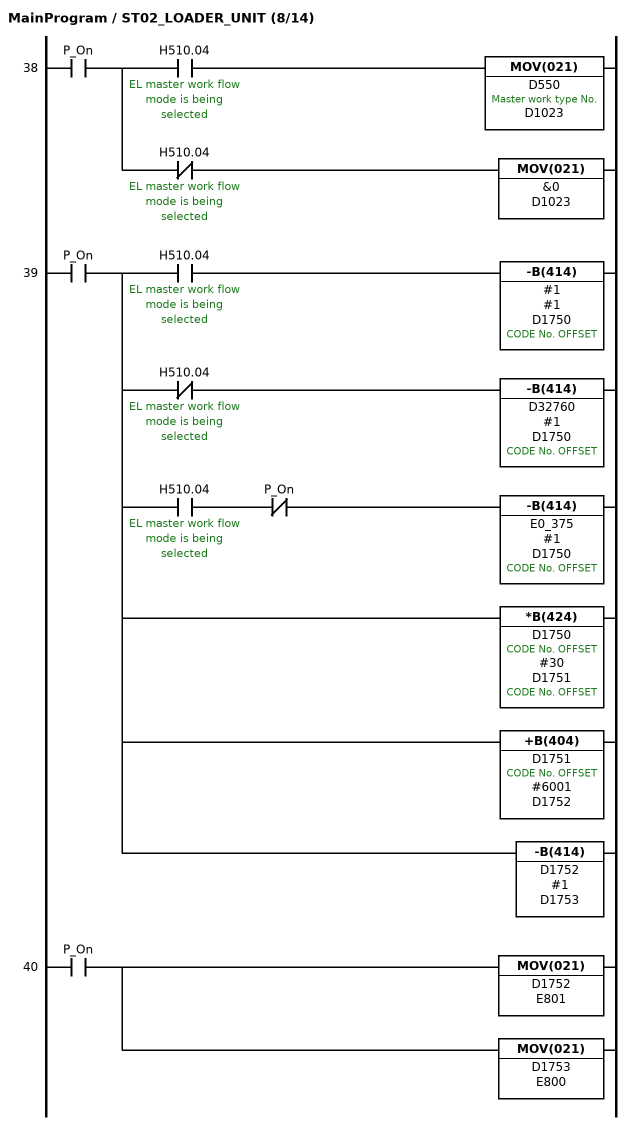
; [picture p312: MainProgram / ST02_LOADER_UNIT, rungs 38-40]
; rung 38
LD P_On
OUT TR0
AND H510.04  ; EL master work flow mode is being selected
MOV(021) D550 D1023  ; Master work type No.
LD TR0
ANDNOT H510.04  ; EL master work flow mode is being selected
MOV(021) &0 D1023
; rung 39
LD P_On
OUT TR0
AND H510.04  ; EL master work flow mode is being selected
-B(414) #1 #1 D1750  ; CODE No. OFFSET
LD TR0
ANDNOT H510.04  ; EL master work flow mode is being selected
-B(414) D32760 #1 D1750  ; CODE No. OFFSET
LD TR0
AND H510.04  ; EL master work flow mode is being selected
ANDNOT P_On
-B(414) E0_375 #1 D1750  ; CODE No. OFFSET
LD TR0
*B(424) D1750 #30 D1751  ; CODE No. OFFSET
+B(404) D1751 #6001 D1752  ; CODE No. OFFSET
-B(414) D1752 #1 D1753
; rung 40
LD P_On
MOV(021) D1752 E801
MOV(021) D1753 E800

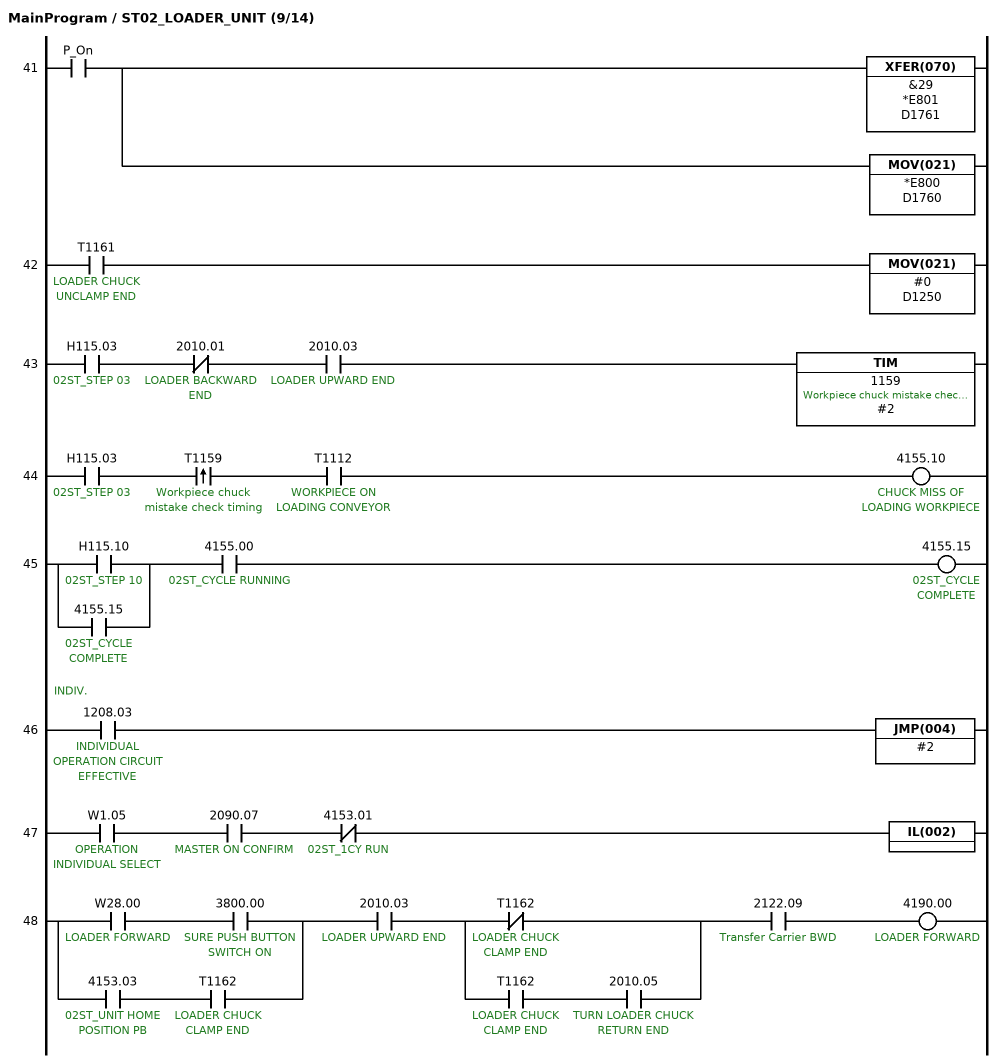
; rung 41
LD P_On
XFER(070) &29 *E801 D1761
MOV(021) *E800 D1760
; rung 42
LD T1161  ; LOADER CHUCK UNCLAMP END
MOV(021) #0 D1250
; rung 43
LD H115.03  ; 02ST_STEP 03
ANDNOT 2010.01  ; LOADER BACKWARD END
AND 2010.03  ; LOADER UPWARD END
TIM 1159 #2  ; Workpiece chuck mistake check timing
; rung 44
LD H115.03  ; 02ST_STEP 03
@AND T1159  ; Workpiece chuck mistake check timing
AND T1112  ; WORKPIECE ON LOADING CONVEYOR
OUT 4155.10  ; CHUCK MISS OF LOADING WORKPIECE
; rung 45
LD H115.10  ; 02ST_STEP 10
OR 4155.15  ; 02ST_CYCLE COMPLETE
AND 4155.00  ; 02ST_CYCLE RUNNING
OUT 4155.15  ; 02ST_CYCLE COMPLETE
; rung 46: INDIV.
LD 1208.03  ; INDIVIDUAL OPERATION CIRCUIT EFFECTIVE
JMP(004) #2
; rung 47
LD W1.05  ; OPERATION INDIVIDUAL SELECT
AND 2090.07  ; MASTER ON CONFIRM
ANDNOT 4153.01  ; 02ST_1CY RUN
IL(002)
; rung 48
LD W28.00  ; LOADER FORWARD
AND 3800.00  ; SURE PUSH BUTTON SWITCH ON
LD 4153.03  ; 02ST_UNIT HOME POSITION PB
AND T1162  ; LOADER CHUCK CLAMP END
ORLD
AND 2010.03  ; LOADER UPWARD END
LDNOT T1162  ; LOADER CHUCK CLAMP END
LD T1162  ; LOADER CHUCK CLAMP END
AND 2010.05  ; TURN LOADER CHUCK RETURN END
ORLD
ANDLD
AND 2122.09  ; Transfer Carrier BWD
OUT 4190.00  ; LOADER FORWARD

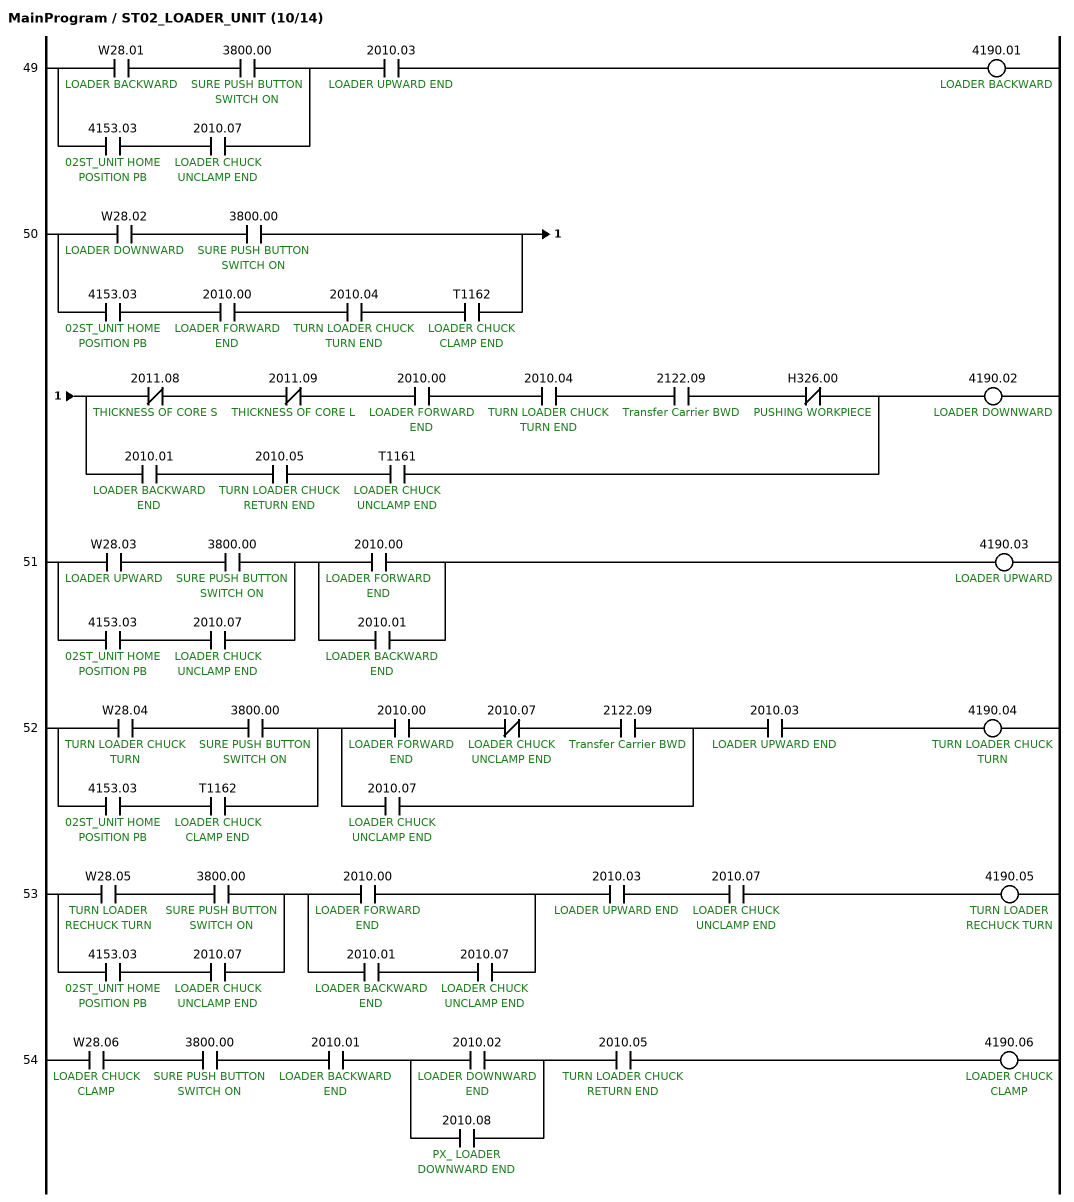
; rung 49
LD W28.01  ; LOADER BACKWARD
AND 3800.00  ; SURE PUSH BUTTON SWITCH ON
LD 4153.03  ; 02ST_UNIT HOME POSITION PB
AND 2010.07  ; LOADER CHUCK UNCLAMP END
ORLD
AND 2010.03  ; LOADER UPWARD END
OUT 4190.01  ; LOADER BACKWARD
; rung 50
LD W28.02  ; LOADER DOWNWARD
AND 3800.00  ; SURE PUSH BUTTON SWITCH ON
LD 4153.03  ; 02ST_UNIT HOME POSITION PB
AND 2010.00  ; LOADER FORWARD END
AND 2010.04  ; TURN LOADER CHUCK TURN END
AND T1162  ; LOADER CHUCK CLAMP END
ORLD
LDNOT 2011.08  ; THICKNESS OF CORE S
ANDNOT 2011.09  ; THICKNESS OF CORE L
AND 2010.00  ; LOADER FORWARD END
AND 2010.04  ; TURN LOADER CHUCK TURN END
AND 2122.09  ; Transfer Carrier BWD
ANDNOT H326.00  ; PUSHING WORKPIECE
LD 2010.01  ; LOADER BACKWARD END
AND 2010.05  ; TURN LOADER CHUCK RETURN END
AND T1161  ; LOADER CHUCK UNCLAMP END
ORLD
ANDLD
OUT 4190.02  ; LOADER DOWNWARD
; rung 51
LD W28.03  ; LOADER UPWARD
AND 3800.00  ; SURE PUSH BUTTON SWITCH ON
LD 4153.03  ; 02ST_UNIT HOME POSITION PB
AND 2010.07  ; LOADER CHUCK UNCLAMP END
ORLD
LD 2010.00  ; LOADER FORWARD END
OR 2010.01  ; LOADER BACKWARD END
ANDLD
OUT 4190.03  ; LOADER UPWARD
; rung 52
LD W28.04  ; TURN LOADER CHUCK TURN
AND 3800.00  ; SURE PUSH BUTTON SWITCH ON
LD 4153.03  ; 02ST_UNIT HOME POSITION PB
AND T1162  ; LOADER CHUCK CLAMP END
ORLD
LD 2010.00  ; LOADER FORWARD END
ANDNOT 2010.07  ; LOADER CHUCK UNCLAMP END
AND 2122.09  ; Transfer Carrier BWD
OR 2010.07  ; LOADER CHUCK UNCLAMP END
ANDLD
AND 2010.03  ; LOADER UPWARD END
OUT 4190.04  ; TURN LOADER CHUCK TURN
; rung 53
LD W28.05  ; TURN LOADER RECHUCK TURN
AND 3800.00  ; SURE PUSH BUTTON SWITCH ON
LD 4153.03  ; 02ST_UNIT HOME POSITION PB
AND 2010.07  ; LOADER CHUCK UNCLAMP END
ORLD
LD 2010.00  ; LOADER FORWARD END
LD 2010.01  ; LOADER BACKWARD END
AND 2010.07  ; LOADER CHUCK UNCLAMP END
ORLD
ANDLD
AND 2010.03  ; LOADER UPWARD END
AND 2010.07  ; LOADER CHUCK UNCLAMP END
OUT 4190.05  ; TURN LOADER RECHUCK TURN
; rung 54
LD W28.06  ; LOADER CHUCK CLAMP
AND 3800.00  ; SURE PUSH BUTTON SWITCH ON
AND 2010.01  ; LOADER BACKWARD END
LD 2010.02  ; LOADER DOWNWARD END
OR 2010.08  ; PX_ LOADER DOWNWARD END
ANDLD
AND 2010.05  ; TURN LOADER CHUCK RETURN END
OUT 4190.06  ; LOADER CHUCK CLAMP

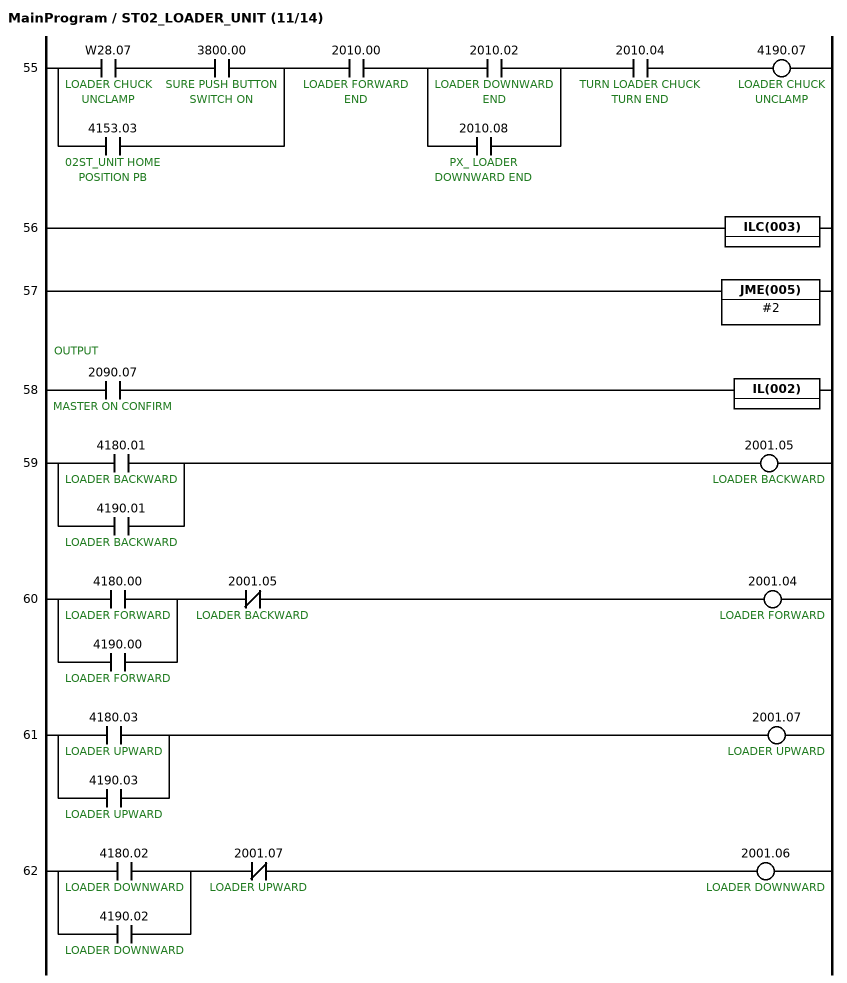
; rung 55
LD W28.07  ; LOADER CHUCK UNCLAMP
AND 3800.00  ; SURE PUSH BUTTON SWITCH ON
OR 4153.03  ; 02ST_UNIT HOME POSITION PB
AND 2010.00  ; LOADER FORWARD END
LD 2010.02  ; LOADER DOWNWARD END
OR 2010.08  ; PX_ LOADER DOWNWARD END
ANDLD
AND 2010.04  ; TURN LOADER CHUCK TURN END
OUT 4190.07  ; LOADER CHUCK UNCLAMP
; rung 56
ILC(003)
; rung 57
JME(005) #2
; rung 58: OUTPUT
LD 2090.07  ; MASTER ON CONFIRM
IL(002)
; rung 59
LD 4180.01  ; LOADER BACKWARD
OR 4190.01  ; LOADER BACKWARD
OUT 2001.05  ; LOADER BACKWARD
; rung 60
LD 4180.00  ; LOADER FORWARD
OR 4190.00  ; LOADER FORWARD
ANDNOT 2001.05  ; LOADER BACKWARD
OUT 2001.04  ; LOADER FORWARD
; rung 61
LD 4180.03  ; LOADER UPWARD
OR 4190.03  ; LOADER UPWARD
OUT 2001.07  ; LOADER UPWARD
; rung 62
LD 4180.02  ; LOADER DOWNWARD
OR 4190.02  ; LOADER DOWNWARD
ANDNOT 2001.07  ; LOADER UPWARD
OUT 2001.06  ; LOADER DOWNWARD

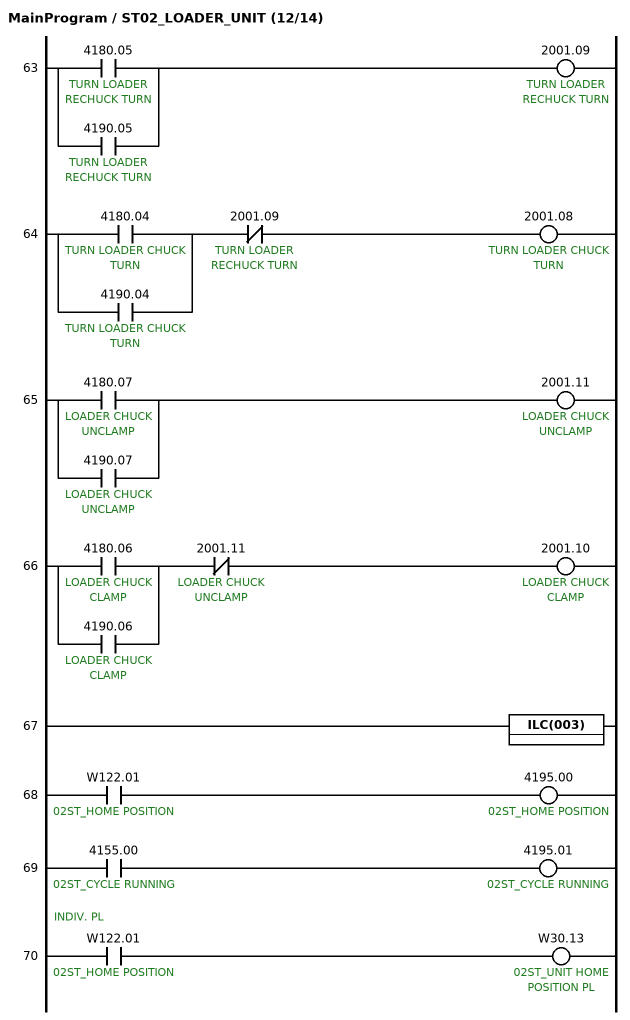
; rung 63
LD 4180.05  ; TURN LOADER RECHUCK TURN
OR 4190.05  ; TURN LOADER RECHUCK TURN
OUT 2001.09  ; TURN LOADER RECHUCK TURN
; rung 64
LD 4180.04  ; TURN LOADER CHUCK TURN
OR 4190.04  ; TURN LOADER CHUCK TURN
ANDNOT 2001.09  ; TURN LOADER RECHUCK TURN
OUT 2001.08  ; TURN LOADER CHUCK TURN
; rung 65
LD 4180.07  ; LOADER CHUCK UNCLAMP
OR 4190.07  ; LOADER CHUCK UNCLAMP
OUT 2001.11  ; LOADER CHUCK UNCLAMP
; rung 66
LD 4180.06  ; LOADER CHUCK CLAMP
OR 4190.06  ; LOADER CHUCK CLAMP
ANDNOT 2001.11  ; LOADER CHUCK UNCLAMP
OUT 2001.10  ; LOADER CHUCK CLAMP
; rung 67
ILC(003)
; rung 68
LD W122.01  ; 02ST_HOME POSITION
OUT 4195.00  ; 02ST_HOME POSITION
; rung 69
LD 4155.00  ; 02ST_CYCLE RUNNING
OUT 4195.01  ; 02ST_CYCLE RUNNING
; rung 70: INDIV. PL
LD W122.01  ; 02ST_HOME POSITION
OUT W30.13  ; 02ST_UNIT HOME POSITION PL

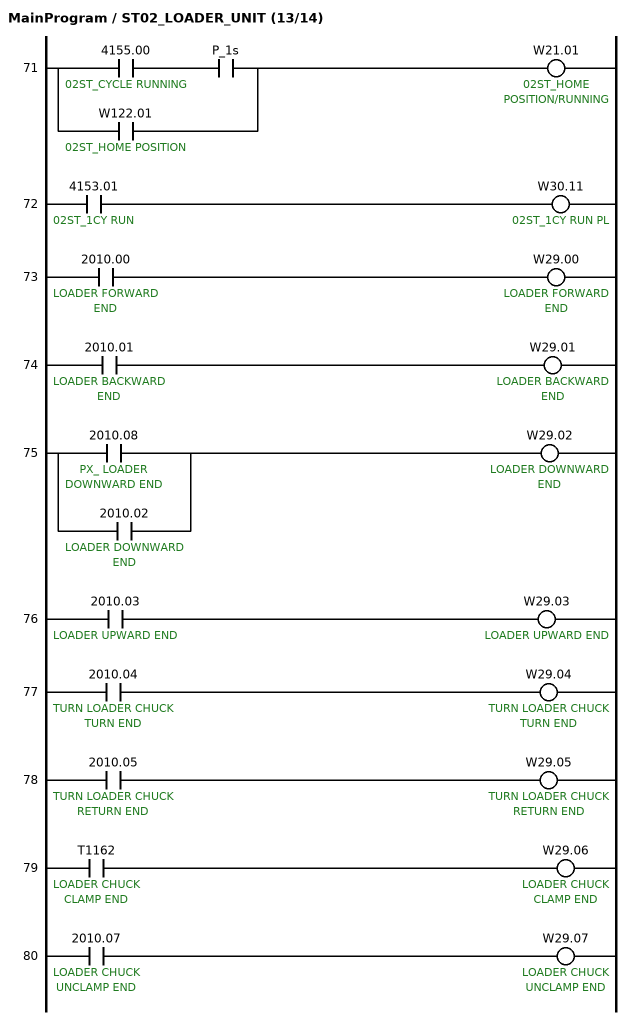
; rung 71
LD 4155.00  ; 02ST_CYCLE RUNNING
AND P_1s
OR W122.01  ; 02ST_HOME POSITION
OUT W21.01  ; 02ST_HOME POSITION/RUNNING
; rung 72
LD 4153.01  ; 02ST_1CY RUN
OUT W30.11  ; 02ST_1CY RUN PL
; rung 73
LD 2010.00  ; LOADER FORWARD END
OUT W29.00  ; LOADER FORWARD END
; rung 74
LD 2010.01  ; LOADER BACKWARD END
OUT W29.01  ; LOADER BACKWARD END
; rung 75
LD 2010.08  ; PX_ LOADER DOWNWARD END
OR 2010.02  ; LOADER DOWNWARD END
OUT W29.02  ; LOADER DOWNWARD END
; rung 76
LD 2010.03  ; LOADER UPWARD END
OUT W29.03  ; LOADER UPWARD END
; rung 77
LD 2010.04  ; TURN LOADER CHUCK TURN END
OUT W29.04  ; TURN LOADER CHUCK TURN END
; rung 78
LD 2010.05  ; TURN LOADER CHUCK RETURN END
OUT W29.05  ; TURN LOADER CHUCK RETURN END
; rung 79
LD T1162  ; LOADER CHUCK CLAMP END
OUT W29.06  ; LOADER CHUCK CLAMP END
; rung 80
LD 2010.07  ; LOADER CHUCK UNCLAMP END
OUT W29.07  ; LOADER CHUCK UNCLAMP END

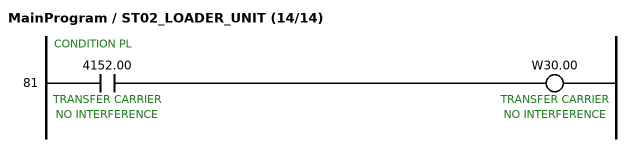
; rung 81: CONDITION PL
LD 4152.00  ; TRANSFER CARRIER NO INTERFERENCE
OUT W30.00  ; TRANSFER CARRIER NO INTERFERENCE

### Section ST03_TRANSFER_CARRIER_UNIT
; rung 0: 03ST_TRANSFER CARRIER UNIT

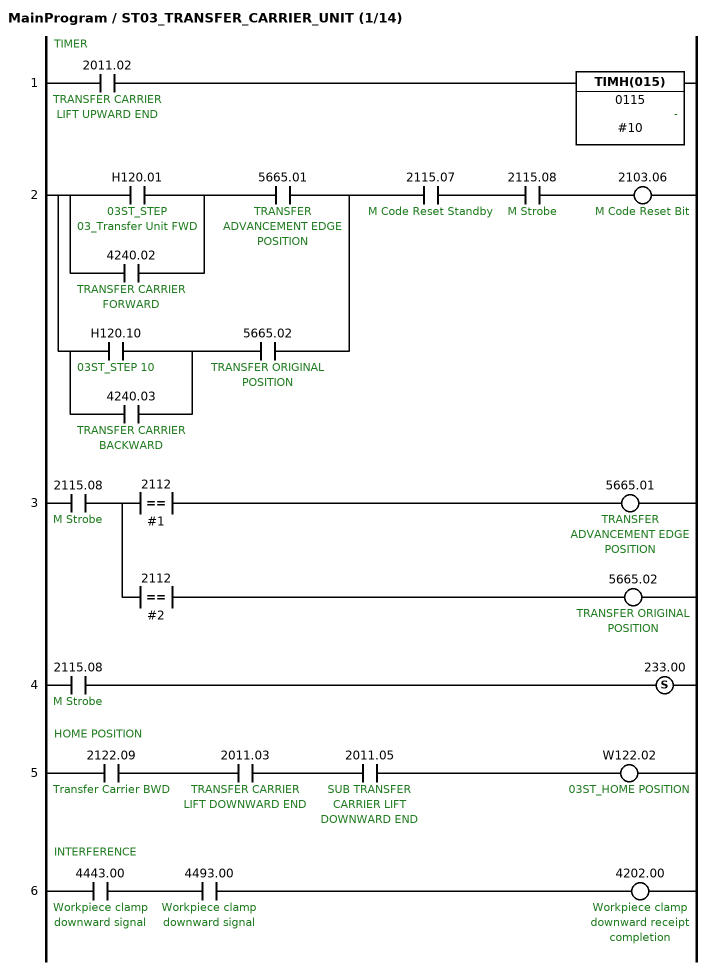
; rung 1: TIMER
LD 2011.02  ; TRANSFER CARRIER LIFT UPWARD END
TIMH(015) 0115 #10  ; -
; rung 2
LD H120.01  ; 03ST_STEP 03_Transfer Unit FWD
OR 4240.02  ; TRANSFER CARRIER FORWARD
AND 5665.01  ; TRANSFER ADVANCEMENT EDGE POSITION
LD H120.10  ; 03ST_STEP 10
OR 4240.03  ; TRANSFER CARRIER BACKWARD
AND 5665.02  ; TRANSFER ORIGINAL POSITION
ORLD
AND 2115.07  ; M Code Reset Standby
AND 2115.08  ; M Strobe
OUT 2103.06  ; M Code Reset Bit
; rung 3
LD 2115.08  ; M Strobe
OUT TR0
AND=(300) 2112 #1
OUT 5665.01  ; TRANSFER ADVANCEMENT EDGE POSITION
LD TR0
AND=(300) 2112 #2
OUT 5665.02  ; TRANSFER ORIGINAL POSITION
; rung 4
LD 2115.08  ; M Strobe
SET 233.00
; rung 5: HOME POSITION
LD 2122.09  ; Transfer Carrier BWD
AND 2011.03  ; TRANSFER CARRIER LIFT DOWNWARD END
AND 2011.05  ; SUB TRANSFER CARRIER LIFT DOWNWARD END
OUT W122.02  ; 03ST_HOME POSITION
; rung 6: INTERFERENCE
LD 4443.00  ; Workpiece clamp downward signal
AND 4493.00  ; Workpiece clamp downward signal
OUT 4202.00  ; Workpiece clamp downward receipt completion

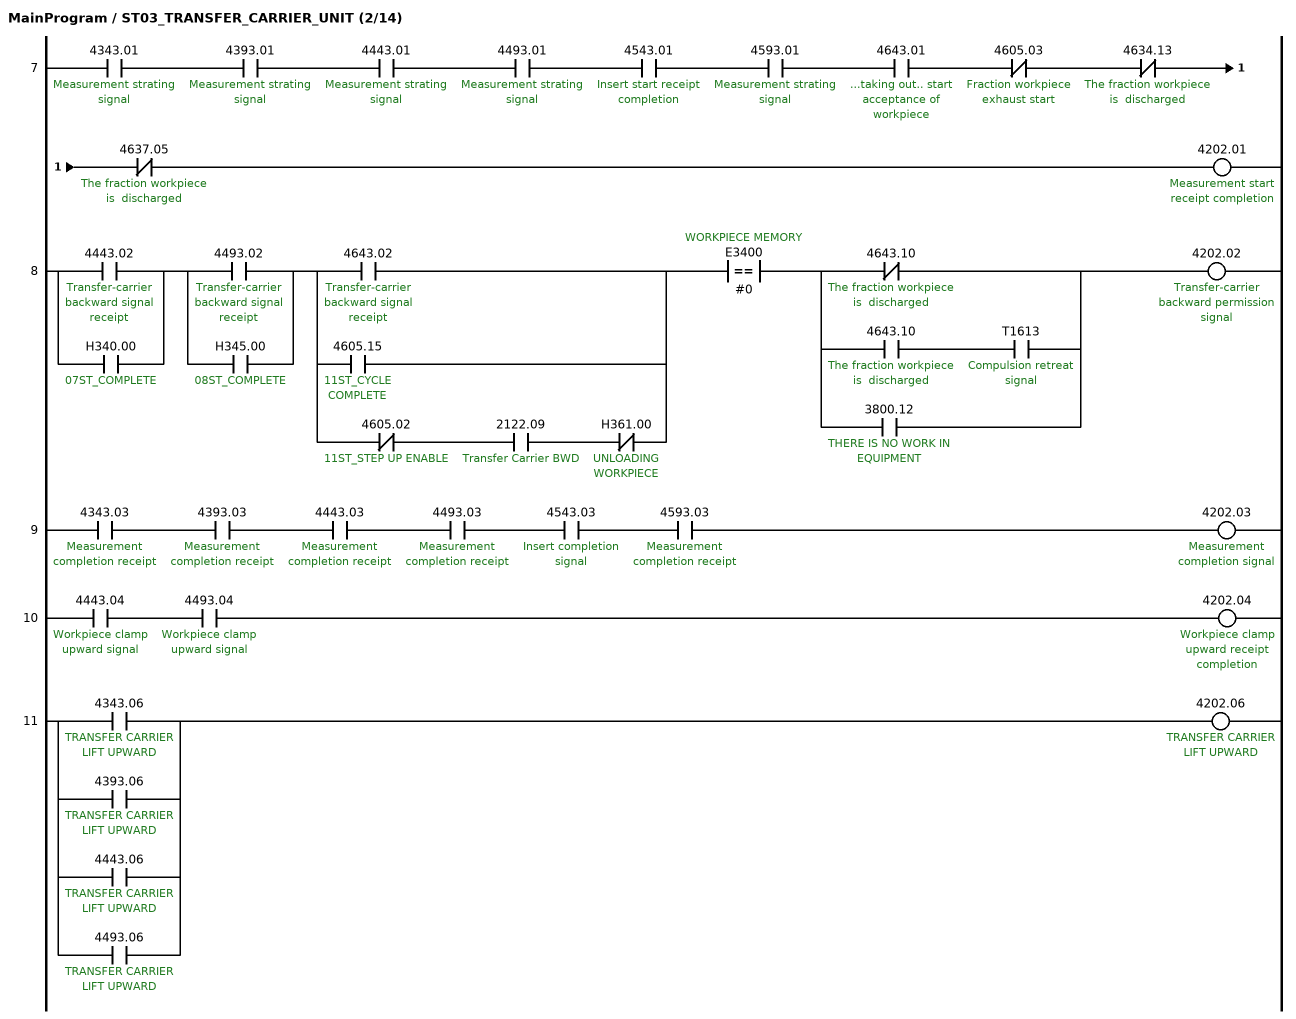
; rung 7
LD 4343.01  ; Measurement strating signal
AND 4393.01  ; Measurement strating signal
AND 4443.01  ; Measurement strating signal
AND 4493.01  ; Measurement strating signal
AND 4543.01  ; Insert start receipt completion
AND 4593.01  ; Measurement strating signal
AND 4643.01  ; ...taking out.. start acceptance of workpiece
ANDNOT 4605.03  ; Fraction workpiece exhaust start
ANDNOT 4634.13  ; The fraction workpiece is  discharged
ANDNOT 4637.05  ; The fraction workpiece is  discharged
OUT 4202.01  ; Measurement start receipt completion
; rung 8
LD 4443.02  ; Transfer-carrier backward signal receipt
OR H340.00  ; 07ST_COMPLETE
LD 4493.02  ; Transfer-carrier backward signal receipt
OR H345.00  ; 08ST_COMPLETE
ANDLD
LD 4643.02  ; Transfer-carrier backward signal receipt
OR 4605.15  ; 11ST_CYCLE COMPLETE
LDNOT 4605.02  ; 11ST_STEP UP ENABLE
AND 2122.09  ; Transfer Carrier BWD
ANDNOT H361.00  ; UNLOADING WORKPIECE
ORLD
ANDLD
AND=(300) E3400 #0  ; WORKPIECE MEMORY
LDNOT 4643.10  ; The fraction workpiece is  discharged
LD 4643.10  ; The fraction workpiece is  discharged
AND T1613  ; Compulsion retreat signal
ORLD
OR 3800.12  ; THERE IS NO WORK IN EQUIPMENT
ANDLD
OUT 4202.02  ; Transfer-carrier backward permission signal
; rung 9
LD 4343.03  ; Measurement completion receipt
AND 4393.03  ; Measurement completion receipt
AND 4443.03  ; Measurement completion receipt
AND 4493.03  ; Measurement completion receipt
AND 4543.03  ; Insert completion signal
AND 4593.03  ; Measurement completion receipt
OUT 4202.03  ; Measurement completion signal
; rung 10
LD 4443.04  ; Workpiece clamp upward signal
AND 4493.04  ; Workpiece clamp upward signal
OUT 4202.04  ; Workpiece clamp upward receipt completion
; rung 11
LD 4343.06  ; TRANSFER CARRIER LIFT UPWARD
OR 4393.06  ; TRANSFER CARRIER LIFT UPWARD
OR 4443.06  ; TRANSFER CARRIER LIFT UPWARD
OR 4493.06  ; TRANSFER CARRIER LIFT UPWARD
OUT 4202.06  ; TRANSFER CARRIER LIFT UPWARD

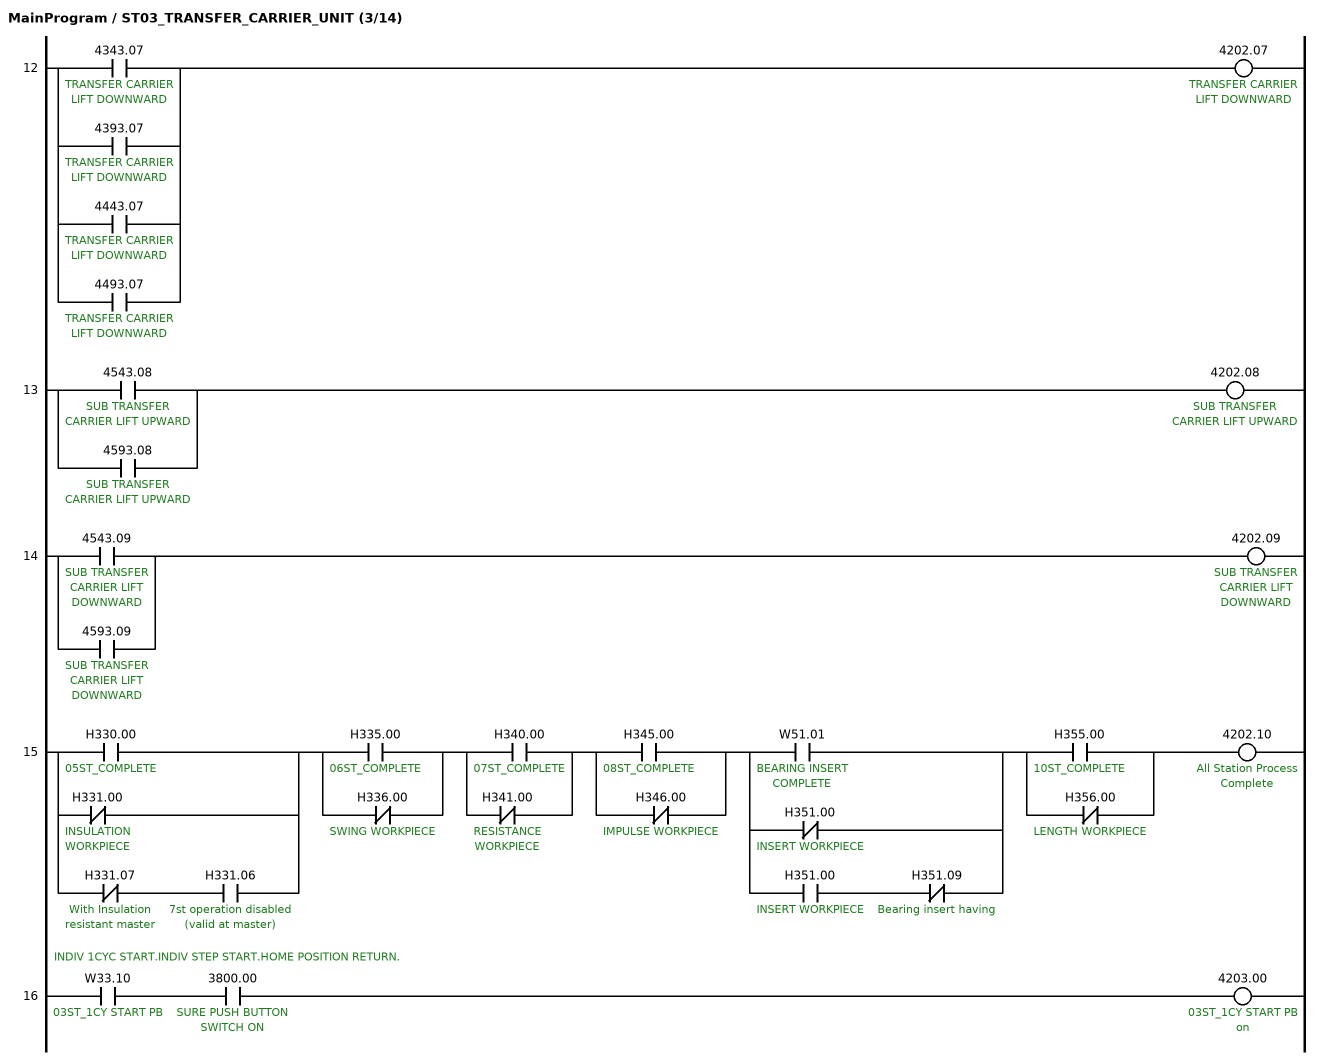
; rung 12
LD 4343.07  ; TRANSFER CARRIER LIFT DOWNWARD
OR 4393.07  ; TRANSFER CARRIER LIFT DOWNWARD
OR 4443.07  ; TRANSFER CARRIER LIFT DOWNWARD
OR 4493.07  ; TRANSFER CARRIER LIFT DOWNWARD
OUT 4202.07  ; TRANSFER CARRIER LIFT DOWNWARD
; rung 13
LD 4543.08  ; SUB TRANSFER CARRIER LIFT UPWARD
OR 4593.08  ; SUB TRANSFER CARRIER LIFT UPWARD
OUT 4202.08  ; SUB TRANSFER CARRIER LIFT UPWARD
; rung 14
LD 4543.09  ; SUB TRANSFER CARRIER LIFT DOWNWARD
OR 4593.09  ; SUB TRANSFER CARRIER LIFT DOWNWARD
OUT 4202.09  ; SUB TRANSFER CARRIER LIFT DOWNWARD
; rung 15
LD H330.00  ; 05ST_COMPLETE
ORNOT H331.00  ; INSULATION WORKPIECE
LDNOT H331.07  ; With Insulation resistant master
AND H331.06  ; 7st operation disabled (valid at master)
ORLD
LD H335.00  ; 06ST_COMPLETE
ORNOT H336.00  ; SWING WORKPIECE
ANDLD
LD H340.00  ; 07ST_COMPLETE
ORNOT H341.00  ; RESISTANCE WORKPIECE
ANDLD
LD H345.00  ; 08ST_COMPLETE
ORNOT H346.00  ; IMPULSE WORKPIECE
ANDLD
LD W51.01  ; BEARING INSERT COMPLETE
ORNOT H351.00  ; INSERT WORKPIECE
LD H351.00  ; INSERT WORKPIECE
ANDNOT H351.09  ; Bearing insert having
ORLD
ANDLD
LD H355.00  ; 10ST_COMPLETE
ORNOT H356.00  ; LENGTH WORKPIECE
ANDLD
OUT 4202.10  ; All Station Process Complete
; rung 16: INDIV 1CYC START.INDIV STEP START.HOME POSITION RETURN.
LD W33.10  ; 03ST_1CY START PB
AND 3800.00  ; SURE PUSH BUTTON SWITCH ON
OUT 4203.00  ; 03ST_1CY START PB on

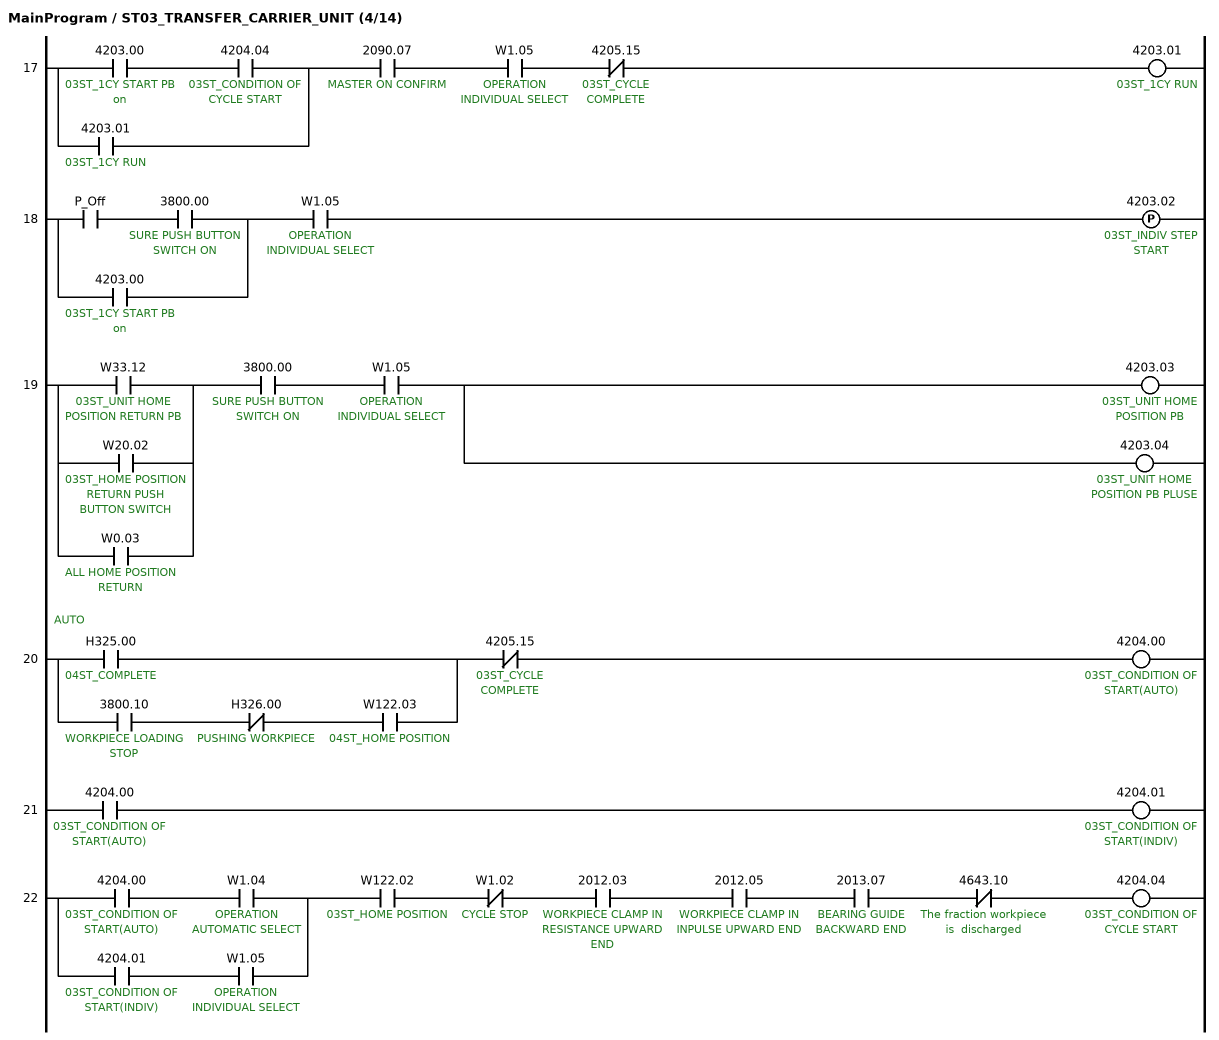
; rung 17
LD 4203.00  ; 03ST_1CY START PB on
AND 4204.04  ; 03ST_CONDITION OF CYCLE START
OR 4203.01  ; 03ST_1CY RUN
AND 2090.07  ; MASTER ON CONFIRM
AND W1.05  ; OPERATION INDIVIDUAL SELECT
ANDNOT 4205.15  ; 03ST_CYCLE COMPLETE
OUT 4203.01  ; 03ST_1CY RUN
; rung 18
LD P_Off
AND 3800.00  ; SURE PUSH BUTTON SWITCH ON
OR 4203.00  ; 03ST_1CY START PB on
AND W1.05  ; OPERATION INDIVIDUAL SELECT
DIFU(013) 4203.02  ; 03ST_INDIV STEP START
; rung 19
LD W33.12  ; 03ST_UNIT HOME POSITION RETURN PB
OR W20.02  ; 03ST_HOME POSITION RETURN PUSH BUTTON SWITCH
OR W0.03  ; ALL HOME POSITION RETURN
AND 3800.00  ; SURE PUSH BUTTON SWITCH ON
AND W1.05  ; OPERATION INDIVIDUAL SELECT
OUT 4203.03  ; 03ST_UNIT HOME POSITION PB
OUT 4203.04  ; 03ST_UNIT HOME POSITION PB PLUSE
; rung 20: AUTO
LD H325.00  ; 04ST_COMPLETE
LD 3800.10  ; WORKPIECE LOADING STOP
ANDNOT H326.00  ; PUSHING WORKPIECE
AND W122.03  ; 04ST_HOME POSITION
ORLD
ANDNOT 4205.15  ; 03ST_CYCLE COMPLETE
OUT 4204.00  ; 03ST_CONDITION OF START(AUTO)
; rung 21
LD 4204.00  ; 03ST_CONDITION OF START(AUTO)
OUT 4204.01  ; 03ST_CONDITION OF START(INDIV)
; rung 22
LD 4204.00  ; 03ST_CONDITION OF START(AUTO)
AND W1.04  ; OPERATION AUTOMATIC SELECT
LD 4204.01  ; 03ST_CONDITION OF START(INDIV)
AND W1.05  ; OPERATION INDIVIDUAL SELECT
ORLD
AND W122.02  ; 03ST_HOME POSITION
ANDNOT W1.02  ; CYCLE STOP
AND 2012.03  ; WORKPIECE CLAMP IN RESISTANCE UPWARD END
AND 2012.05  ; WORKPIECE CLAMP IN INPULSE UPWARD END
AND 2013.07  ; BEARING GUIDE BACKWARD END
ANDNOT 4643.10  ; The fraction workpiece is  discharged
OUT 4204.04  ; 03ST_CONDITION OF CYCLE START

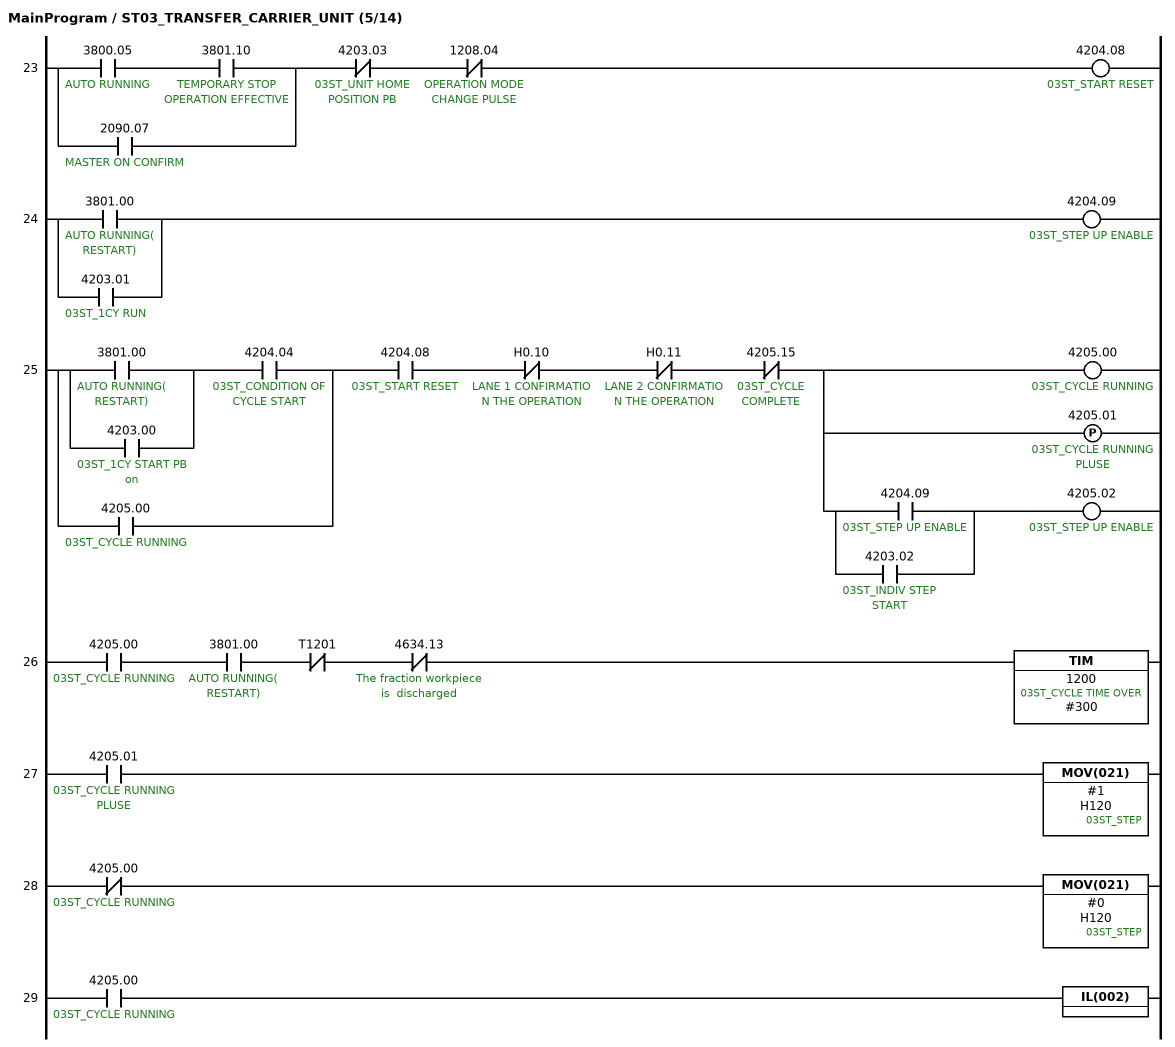
; rung 23
LD 3800.05  ; AUTO RUNNING
AND 3801.10  ; TEMPORARY STOP OPERATION EFFECTIVE
OR 2090.07  ; MASTER ON CONFIRM
ANDNOT 4203.03  ; 03ST_UNIT HOME POSITION PB
ANDNOT 1208.04  ; OPERATION MODE CHANGE PULSE
OUT 4204.08  ; 03ST_START RESET
; rung 24
LD 3801.00  ; AUTO RUNNING(RESTART)
OR 4203.01  ; 03ST_1CY RUN
OUT 4204.09  ; 03ST_STEP UP ENABLE
; rung 25
LD 3801.00  ; AUTO RUNNING(RESTART)
OR 4203.00  ; 03ST_1CY START PB on
AND 4204.04  ; 03ST_CONDITION OF CYCLE START
OR 4205.00  ; 03ST_CYCLE RUNNING
AND 4204.08  ; 03ST_START RESET
ANDNOT H0.10  ; LANE 1 CONFIRMATION THE OPERATION
ANDNOT H0.11  ; LANE 2 CONFIRMATION THE OPERATION
ANDNOT 4205.15  ; 03ST_CYCLE COMPLETE
OUT 4205.00  ; 03ST_CYCLE RUNNING
DIFU(013) 4205.01  ; 03ST_CYCLE RUNNING PLUSE
LD 4204.09  ; 03ST_STEP UP ENABLE
OR 4203.02  ; 03ST_INDIV STEP START
ANDLD
OUT 4205.02  ; 03ST_STEP UP ENABLE
; rung 26
LD 4205.00  ; 03ST_CYCLE RUNNING
AND 3801.00  ; AUTO RUNNING(RESTART)
ANDNOT T1201
ANDNOT 4634.13  ; The fraction workpiece is  discharged
TIM 1200 #300  ; 03ST_CYCLE TIME OVER
; rung 27
LD 4205.01  ; 03ST_CYCLE RUNNING PLUSE
MOV(021) #1 H120  ; 03ST_STEP
; rung 28
LDNOT 4205.00  ; 03ST_CYCLE RUNNING
MOV(021) #0 H120  ; 03ST_STEP
; rung 29
LD 4205.00  ; 03ST_CYCLE RUNNING
IL(002)

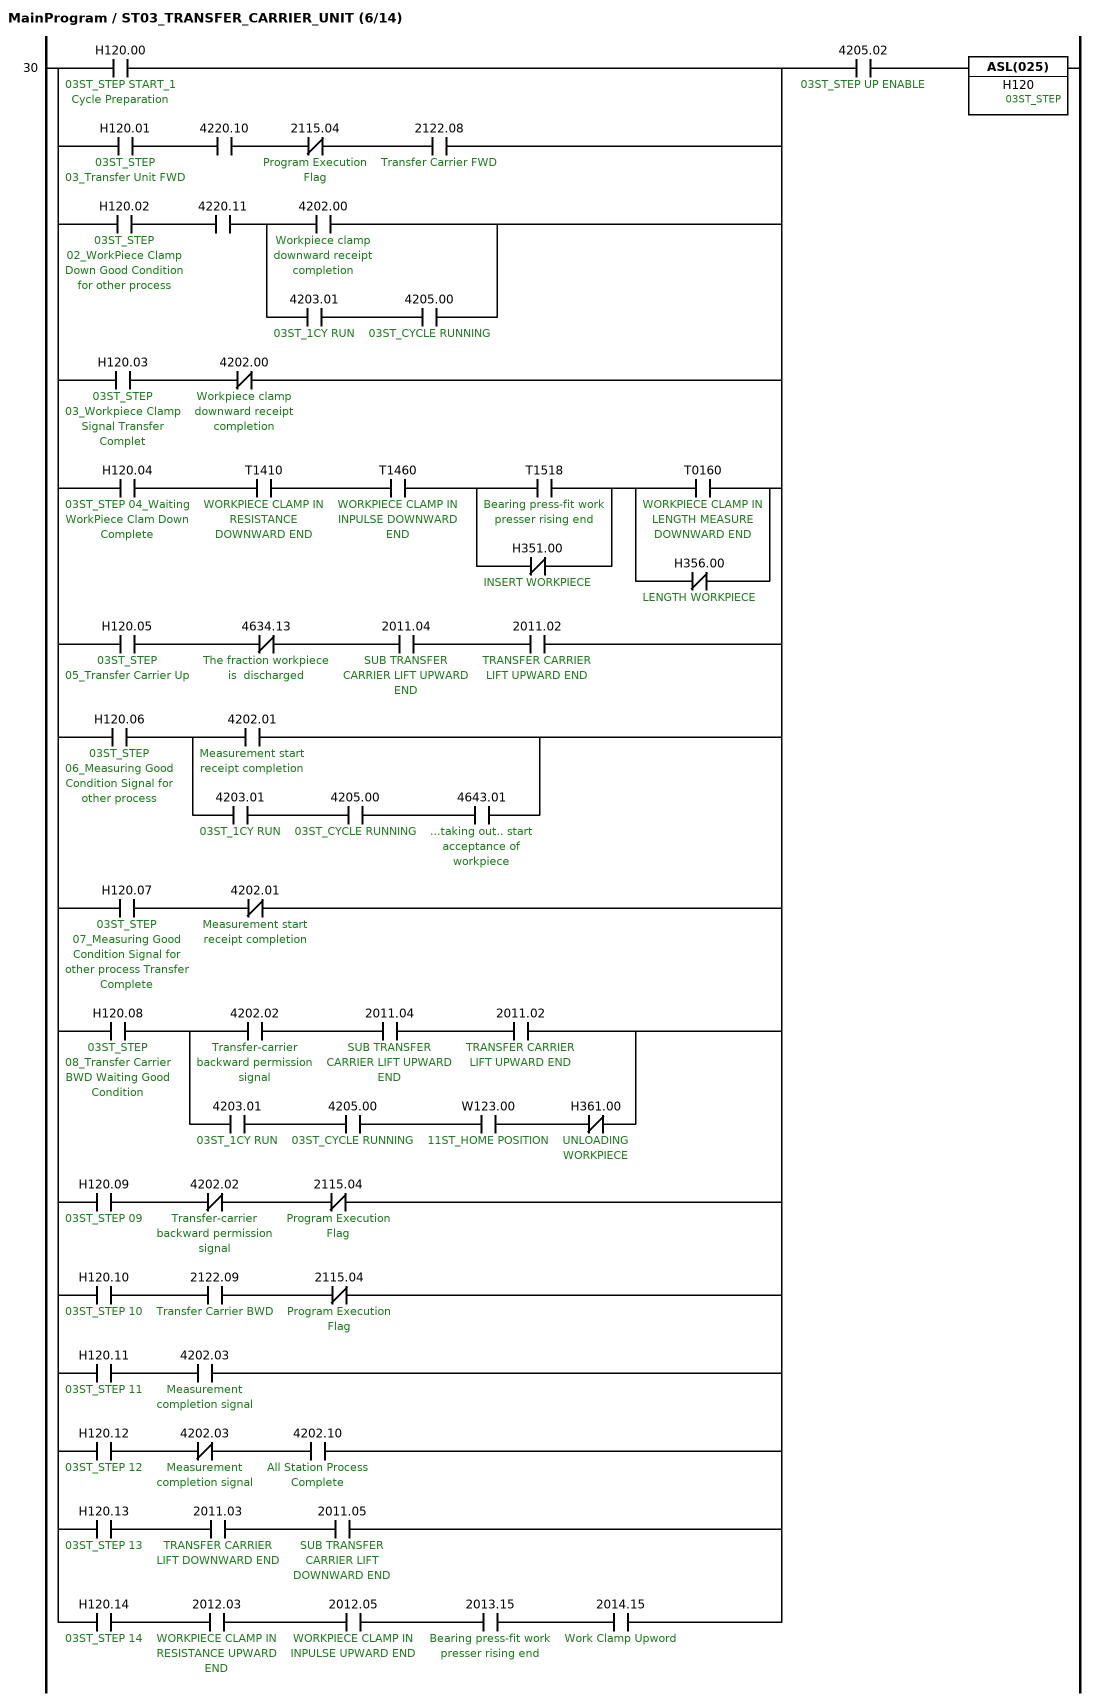
; rung 30
LD H120.00  ; 03ST_STEP START_1 Cycle Preparation
LD H120.01  ; 03ST_STEP 03_Transfer Unit FWD
AND 4220.10
ANDNOT 2115.04  ; Program Execution Flag
AND 2122.08  ; Transfer Carrier FWD
ORLD
LD H120.02  ; 03ST_STEP 02_WorkPiece Clamp Down Good Condition for other process
AND 4220.11
LD 4202.00  ; Workpiece clamp downward receipt completion
LD 4203.01  ; 03ST_1CY RUN
AND 4205.00  ; 03ST_CYCLE RUNNING
ORLD
ANDLD
ORLD
LD H120.03  ; 03ST_STEP 03_Workpiece Clamp Signal Transfer Complet
ANDNOT 4202.00  ; Workpiece clamp downward receipt completion
ORLD
LD H120.04  ; 03ST_STEP 04_Waiting WorkPiece Clam Down Complete
AND T1410  ; WORKPIECE CLAMP IN RESISTANCE DOWNWARD END
AND T1460  ; WORKPIECE CLAMP IN INPULSE DOWNWARD END
LD T1518  ; Bearing press-fit work presser rising end
ORNOT H351.00  ; INSERT WORKPIECE
ANDLD
LD T0160  ; WORKPIECE CLAMP IN LENGTH MEASURE DOWNWARD END
ORNOT H356.00  ; LENGTH WORKPIECE
ANDLD
ORLD
LD H120.05  ; 03ST_STEP 05_Transfer Carrier Up
ANDNOT 4634.13  ; The fraction workpiece is  discharged
AND 2011.04  ; SUB TRANSFER CARRIER LIFT UPWARD END
AND 2011.02  ; TRANSFER CARRIER LIFT UPWARD END
ORLD
LD H120.06  ; 03ST_STEP 06_Measuring Good Condition Signal for other process
LD 4202.01  ; Measurement start receipt completion
LD 4203.01  ; 03ST_1CY RUN
AND 4205.00  ; 03ST_CYCLE RUNNING
AND 4643.01  ; ...taking out.. start acceptance of workpiece
ORLD
ANDLD
ORLD
LD H120.07  ; 03ST_STEP 07_Measuring Good Condition Signal for other process Transfer Complete
ANDNOT 4202.01  ; Measurement start receipt completion
ORLD
LD H120.08  ; 03ST_STEP 08_Transfer Carrier BWD Waiting Good Condition
LD 4202.02  ; Transfer-carrier backward permission signal
AND 2011.04  ; SUB TRANSFER CARRIER LIFT UPWARD END
AND 2011.02  ; TRANSFER CARRIER LIFT UPWARD END
LD 4203.01  ; 03ST_1CY RUN
AND 4205.00  ; 03ST_CYCLE RUNNING
AND W123.00  ; 11ST_HOME POSITION
ANDNOT H361.00  ; UNLOADING WORKPIECE
ORLD
ANDLD
ORLD
LD H120.09  ; 03ST_STEP 09
ANDNOT 4202.02  ; Transfer-carrier backward permission signal
ANDNOT 2115.04  ; Program Execution Flag
ORLD
LD H120.10  ; 03ST_STEP 10
AND 2122.09  ; Transfer Carrier BWD
ANDNOT 2115.04  ; Program Execution Flag
ORLD
LD H120.11  ; 03ST_STEP 11
AND 4202.03  ; Measurement completion signal
ORLD
LD H120.12  ; 03ST_STEP 12
ANDNOT 4202.03  ; Measurement completion signal
AND 4202.10  ; All Station Process Complete
ORLD
LD H120.13  ; 03ST_STEP 13
AND 2011.03  ; TRANSFER CARRIER LIFT DOWNWARD END
AND 2011.05  ; SUB TRANSFER CARRIER LIFT DOWNWARD END
ORLD
LD H120.14  ; 03ST_STEP 14
AND 2012.03  ; WORKPIECE CLAMP IN RESISTANCE UPWARD END
AND 2012.05  ; WORKPIECE CLAMP IN INPULSE UPWARD END
AND 2013.15  ; Bearing press-fit work presser rising end
AND 2014.15  ; Work Clamp Upword
ORLD
AND 4205.02  ; 03ST_STEP UP ENABLE
ASL(025) H120  ; 03ST_STEP

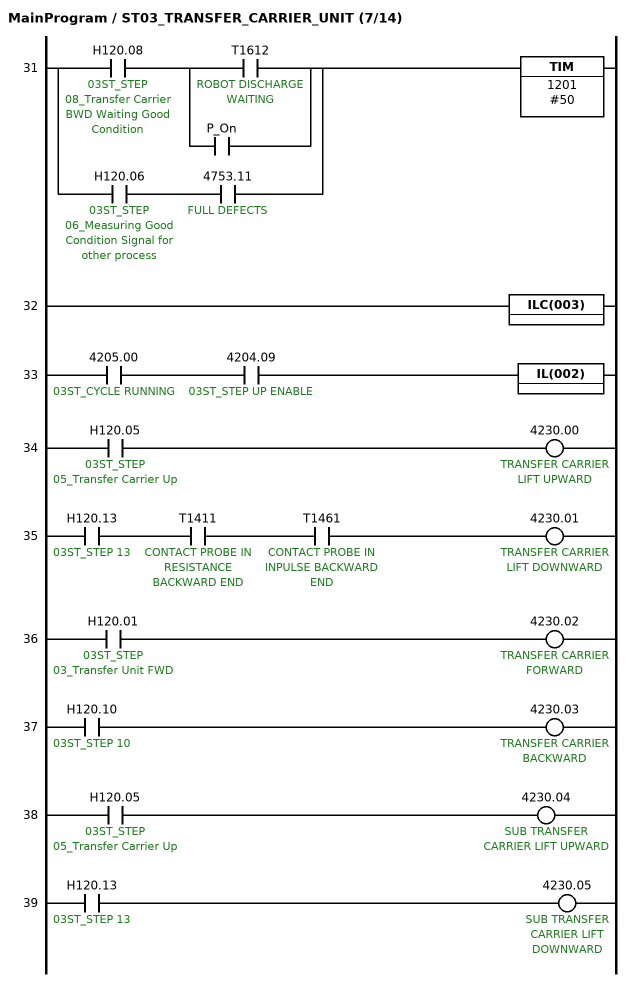
; rung 31
LD H120.08  ; 03ST_STEP 08_Transfer Carrier BWD Waiting Good Condition
LD T1612  ; ROBOT DISCHARGE WAITING
OR P_On
ANDLD
LD H120.06  ; 03ST_STEP 06_Measuring Good Condition Signal for other process
AND 4753.11  ; FULL DEFECTS
ORLD
TIM 1201 #50
; rung 32
ILC(003)
; rung 33
LD 4205.00  ; 03ST_CYCLE RUNNING
AND 4204.09  ; 03ST_STEP UP ENABLE
IL(002)
; rung 34
LD H120.05  ; 03ST_STEP 05_Transfer Carrier Up
OUT 4230.00  ; TRANSFER CARRIER LIFT UPWARD
; rung 35
LD H120.13  ; 03ST_STEP 13
AND T1411  ; CONTACT PROBE IN RESISTANCE BACKWARD END
AND T1461  ; CONTACT PROBE IN INPULSE BACKWARD END
OUT 4230.01  ; TRANSFER CARRIER LIFT DOWNWARD
; rung 36
LD H120.01  ; 03ST_STEP 03_Transfer Unit FWD
OUT 4230.02  ; TRANSFER CARRIER FORWARD
; rung 37
LD H120.10  ; 03ST_STEP 10
OUT 4230.03  ; TRANSFER CARRIER BACKWARD
; rung 38
LD H120.05  ; 03ST_STEP 05_Transfer Carrier Up
OUT 4230.04  ; SUB TRANSFER CARRIER LIFT UPWARD
; rung 39
LD H120.13  ; 03ST_STEP 13
OUT 4230.05  ; SUB TRANSFER CARRIER LIFT DOWNWARD

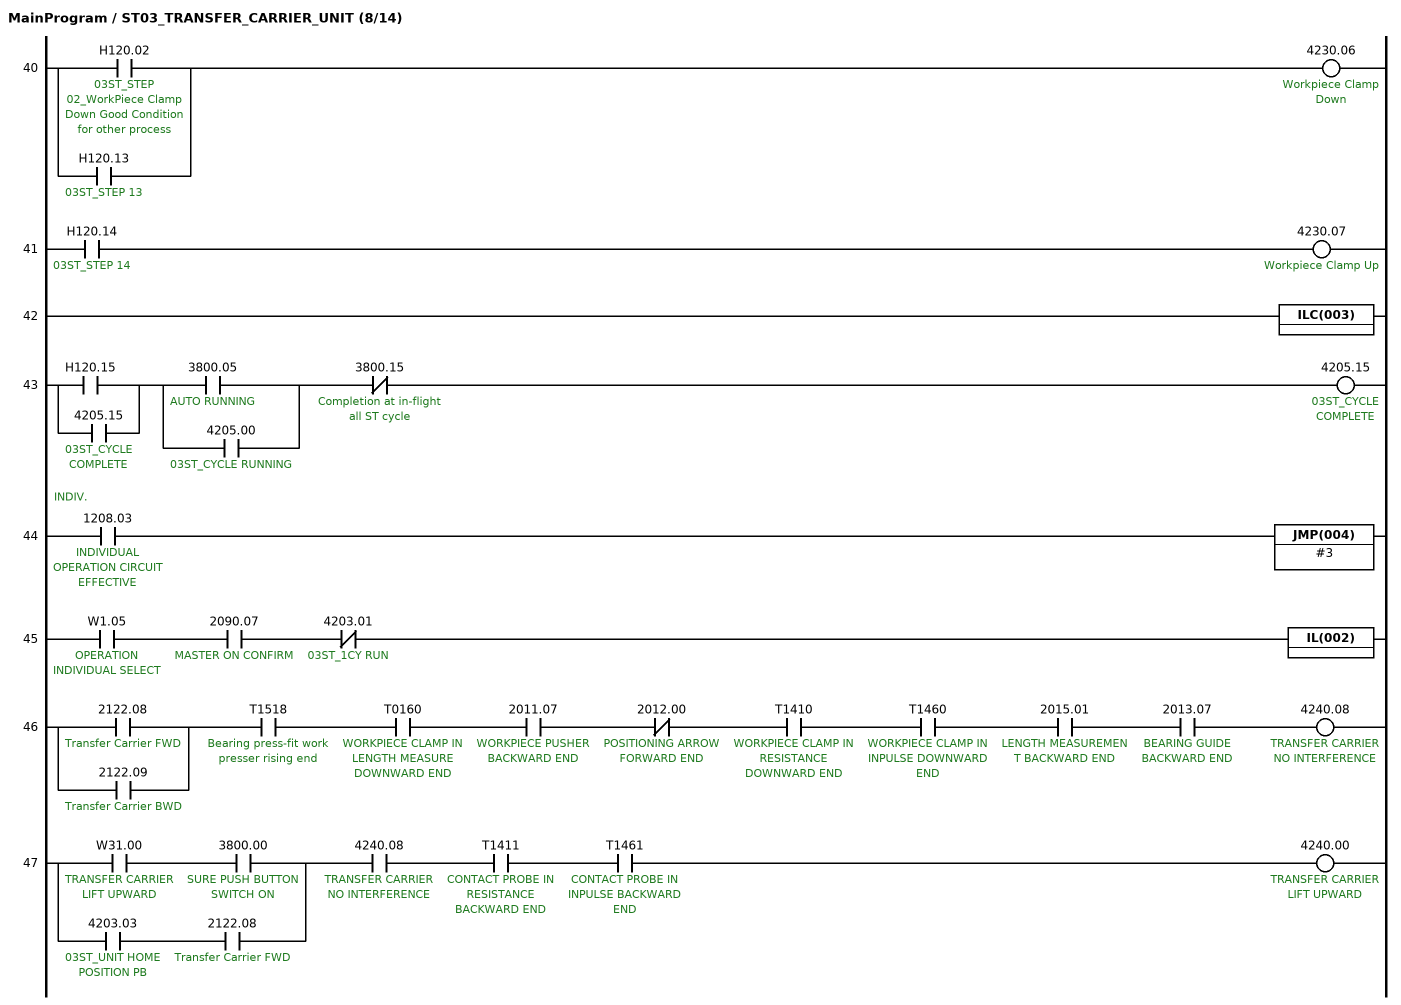
; rung 40
LD H120.02  ; 03ST_STEP 02_WorkPiece Clamp Down Good Condition for other process
OR H120.13  ; 03ST_STEP 13
OUT 4230.06  ; Workpiece Clamp Down
; rung 41
LD H120.14  ; 03ST_STEP 14
OUT 4230.07  ; Workpiece Clamp Up
; rung 42
ILC(003)
; rung 43
LD H120.15
OR 4205.15  ; 03ST_CYCLE COMPLETE
LD 3800.05  ; AUTO RUNNING
OR 4205.00  ; 03ST_CYCLE RUNNING
ANDLD
ANDNOT 3800.15  ; Completion at in-flight all ST cycle
OUT 4205.15  ; 03ST_CYCLE COMPLETE
; rung 44: INDIV.
LD 1208.03  ; INDIVIDUAL OPERATION CIRCUIT EFFECTIVE
JMP(004) #3
; rung 45
LD W1.05  ; OPERATION INDIVIDUAL SELECT
AND 2090.07  ; MASTER ON CONFIRM
ANDNOT 4203.01  ; 03ST_1CY RUN
IL(002)
; rung 46
LD 2122.08  ; Transfer Carrier FWD
OR 2122.09  ; Transfer Carrier BWD
AND T1518  ; Bearing press-fit work presser rising end
AND T0160  ; WORKPIECE CLAMP IN LENGTH MEASURE DOWNWARD END
AND 2011.07  ; WORKPIECE PUSHER BACKWARD END
ANDNOT 2012.00  ; POSITIONING ARROW FORWARD END
AND T1410  ; WORKPIECE CLAMP IN RESISTANCE DOWNWARD END
AND T1460  ; WORKPIECE CLAMP IN INPULSE DOWNWARD END
AND 2015.01  ; LENGTH MEASUREMENT BACKWARD END
AND 2013.07  ; BEARING GUIDE BACKWARD END
OUT 4240.08  ; TRANSFER CARRIER NO INTERFERENCE
; rung 47
LD W31.00  ; TRANSFER CARRIER LIFT UPWARD
AND 3800.00  ; SURE PUSH BUTTON SWITCH ON
LD 4203.03  ; 03ST_UNIT HOME POSITION PB
AND 2122.08  ; Transfer Carrier FWD
ORLD
AND 4240.08  ; TRANSFER CARRIER NO INTERFERENCE
AND T1411  ; CONTACT PROBE IN RESISTANCE BACKWARD END
AND T1461  ; CONTACT PROBE IN INPULSE BACKWARD END
OUT 4240.00  ; TRANSFER CARRIER LIFT UPWARD

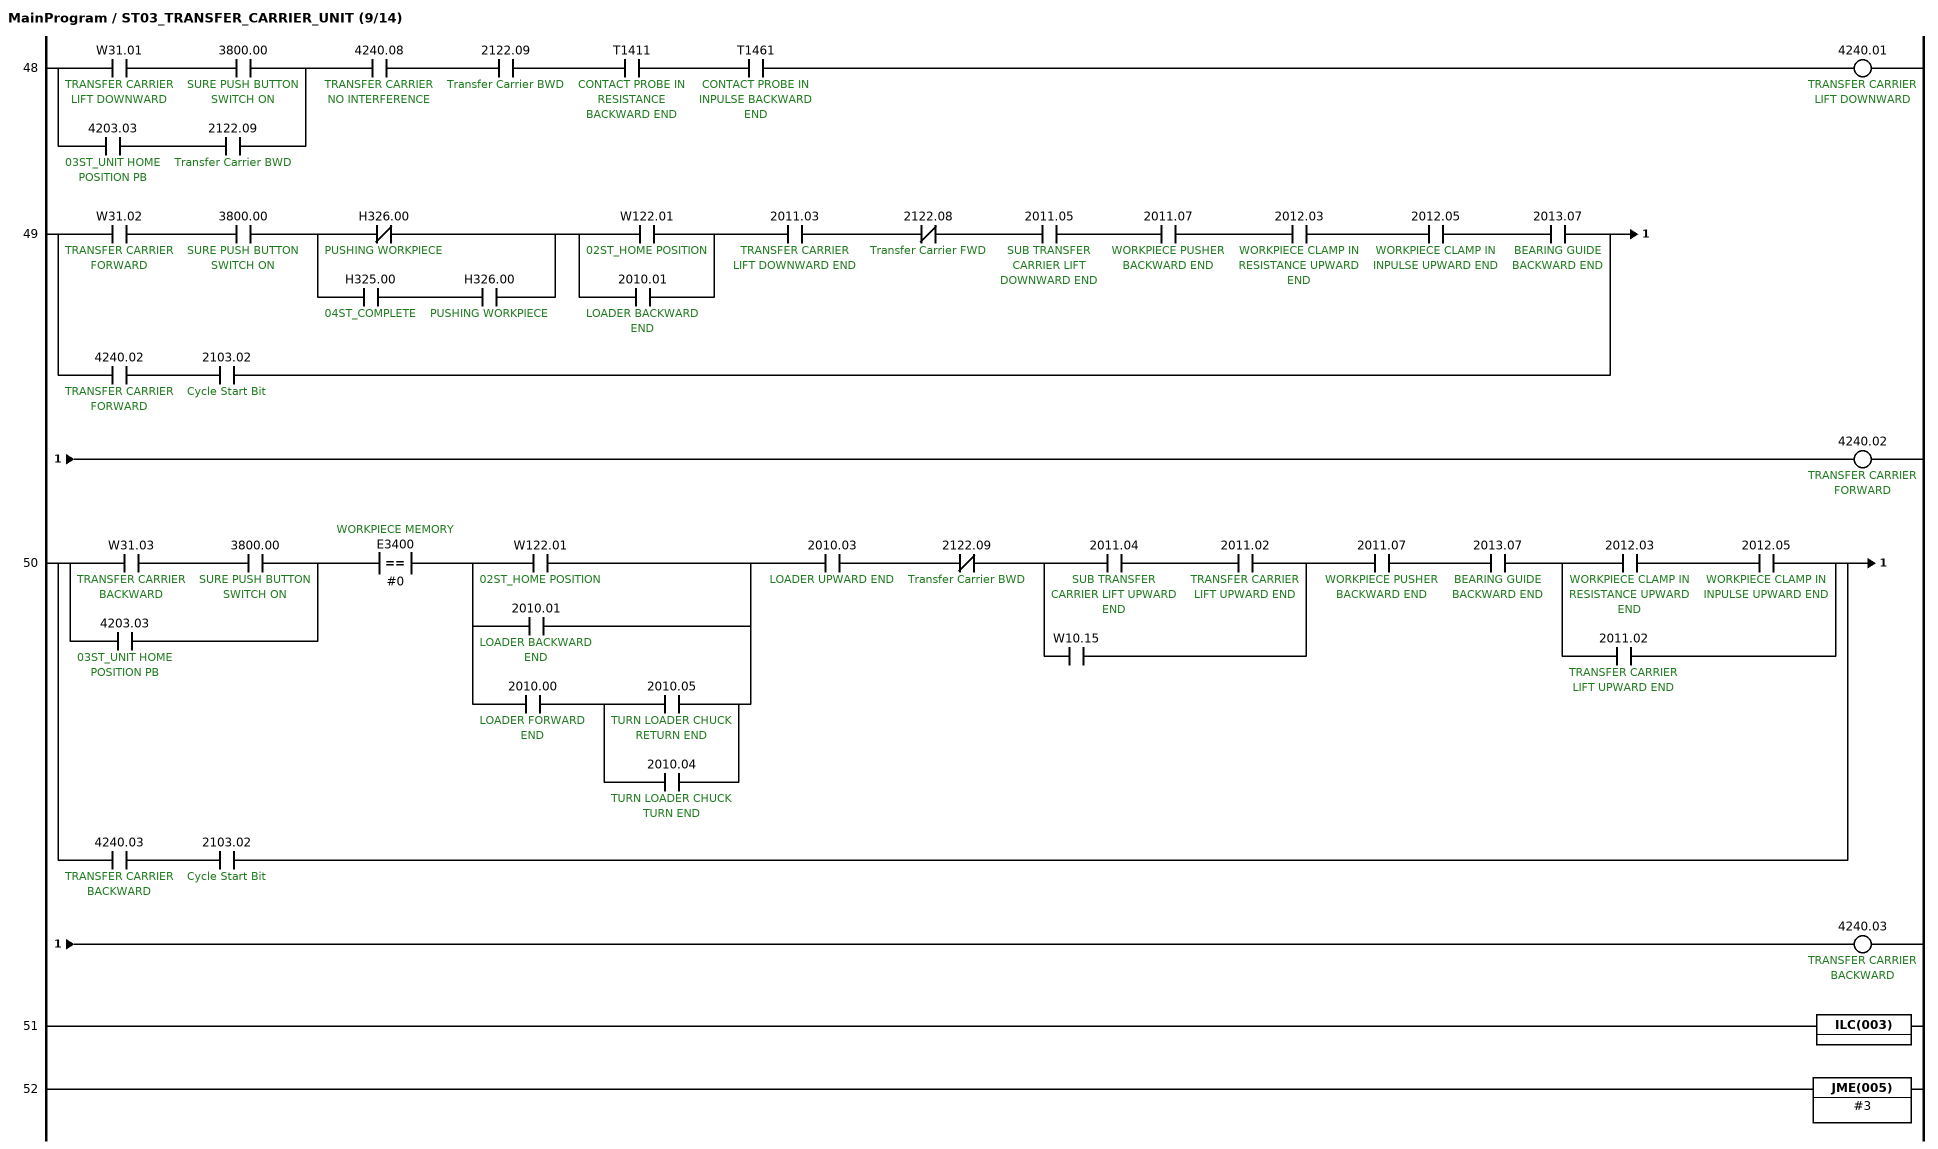
; rung 48
LD W31.01  ; TRANSFER CARRIER LIFT DOWNWARD
AND 3800.00  ; SURE PUSH BUTTON SWITCH ON
LD 4203.03  ; 03ST_UNIT HOME POSITION PB
AND 2122.09  ; Transfer Carrier BWD
ORLD
AND 4240.08  ; TRANSFER CARRIER NO INTERFERENCE
AND 2122.09  ; Transfer Carrier BWD
AND T1411  ; CONTACT PROBE IN RESISTANCE BACKWARD END
AND T1461  ; CONTACT PROBE IN INPULSE BACKWARD END
OUT 4240.01  ; TRANSFER CARRIER LIFT DOWNWARD
; rung 49
LD W31.02  ; TRANSFER CARRIER FORWARD
AND 3800.00  ; SURE PUSH BUTTON SWITCH ON
LDNOT H326.00  ; PUSHING WORKPIECE
LD H325.00  ; 04ST_COMPLETE
AND H326.00  ; PUSHING WORKPIECE
ORLD
ANDLD
LD W122.01  ; 02ST_HOME POSITION
OR 2010.01  ; LOADER BACKWARD END
ANDLD
AND 2011.03  ; TRANSFER CARRIER LIFT DOWNWARD END
ANDNOT 2122.08  ; Transfer Carrier FWD
AND 2011.05  ; SUB TRANSFER CARRIER LIFT DOWNWARD END
AND 2011.07  ; WORKPIECE PUSHER BACKWARD END
AND 2012.03  ; WORKPIECE CLAMP IN RESISTANCE UPWARD END
AND 2012.05  ; WORKPIECE CLAMP IN INPULSE UPWARD END
AND 2013.07  ; BEARING GUIDE BACKWARD END
LD 4240.02  ; TRANSFER CARRIER FORWARD
AND 2103.02  ; Cycle Start Bit
ORLD
OUT 4240.02  ; TRANSFER CARRIER FORWARD
; rung 50
LD W31.03  ; TRANSFER CARRIER BACKWARD
AND 3800.00  ; SURE PUSH BUTTON SWITCH ON
OR 4203.03  ; 03ST_UNIT HOME POSITION PB
AND=(300) E3400 #0  ; WORKPIECE MEMORY
LD W122.01  ; 02ST_HOME POSITION
OR 2010.01  ; LOADER BACKWARD END
LD 2010.00  ; LOADER FORWARD END
LD 2010.05  ; TURN LOADER CHUCK RETURN END
OR 2010.04  ; TURN LOADER CHUCK TURN END
ANDLD
ORLD
ANDLD
AND 2010.03  ; LOADER UPWARD END
ANDNOT 2122.09  ; Transfer Carrier BWD
LD 2011.04  ; SUB TRANSFER CARRIER LIFT UPWARD END
AND 2011.02  ; TRANSFER CARRIER LIFT UPWARD END
OR W10.15
ANDLD
AND 2011.07  ; WORKPIECE PUSHER BACKWARD END
AND 2013.07  ; BEARING GUIDE BACKWARD END
LD 2012.03  ; WORKPIECE CLAMP IN RESISTANCE UPWARD END
AND 2012.05  ; WORKPIECE CLAMP IN INPULSE UPWARD END
OR 2011.02  ; TRANSFER CARRIER LIFT UPWARD END
ANDLD
LD 4240.03  ; TRANSFER CARRIER BACKWARD
AND 2103.02  ; Cycle Start Bit
ORLD
OUT 4240.03  ; TRANSFER CARRIER BACKWARD
; rung 51
ILC(003)
; rung 52
JME(005) #3

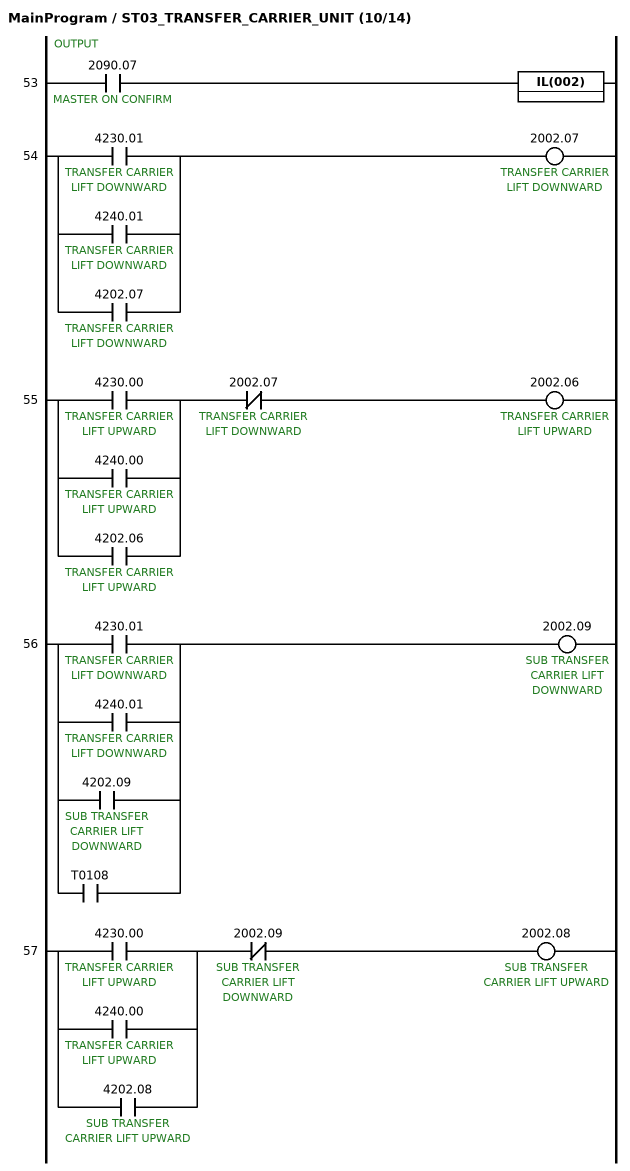
; rung 53: OUTPUT
LD 2090.07  ; MASTER ON CONFIRM
IL(002)
; rung 54
LD 4230.01  ; TRANSFER CARRIER LIFT DOWNWARD
OR 4240.01  ; TRANSFER CARRIER LIFT DOWNWARD
OR 4202.07  ; TRANSFER CARRIER LIFT DOWNWARD
OUT 2002.07  ; TRANSFER CARRIER LIFT DOWNWARD
; rung 55
LD 4230.00  ; TRANSFER CARRIER LIFT UPWARD
OR 4240.00  ; TRANSFER CARRIER LIFT UPWARD
OR 4202.06  ; TRANSFER CARRIER LIFT UPWARD
ANDNOT 2002.07  ; TRANSFER CARRIER LIFT DOWNWARD
OUT 2002.06  ; TRANSFER CARRIER LIFT UPWARD
; rung 56
LD 4230.01  ; TRANSFER CARRIER LIFT DOWNWARD
OR 4240.01  ; TRANSFER CARRIER LIFT DOWNWARD
OR 4202.09  ; SUB TRANSFER CARRIER LIFT DOWNWARD
OR T0108
OUT 2002.09  ; SUB TRANSFER CARRIER LIFT DOWNWARD
; rung 57
LD 4230.00  ; TRANSFER CARRIER LIFT UPWARD
OR 4240.00  ; TRANSFER CARRIER LIFT UPWARD
OR 4202.08  ; SUB TRANSFER CARRIER LIFT UPWARD
ANDNOT 2002.09  ; SUB TRANSFER CARRIER LIFT DOWNWARD
OUT 2002.08  ; SUB TRANSFER CARRIER LIFT UPWARD

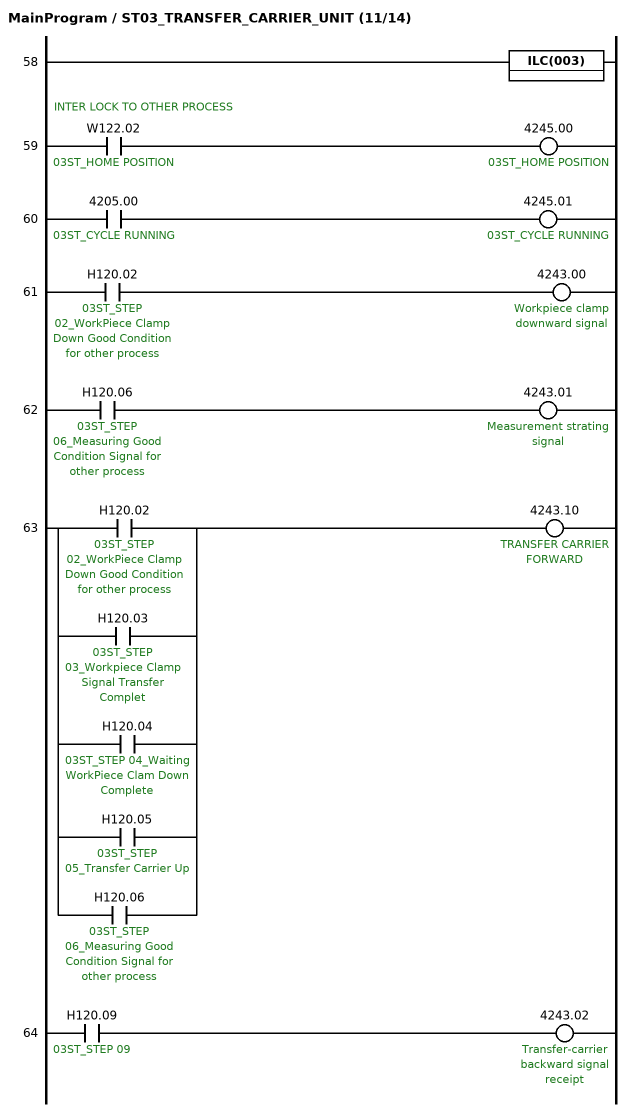
; rung 58
ILC(003)
; rung 59: INTER LOCK TO OTHER PROCESS
LD W122.02  ; 03ST_HOME POSITION
OUT 4245.00  ; 03ST_HOME POSITION
; rung 60
LD 4205.00  ; 03ST_CYCLE RUNNING
OUT 4245.01  ; 03ST_CYCLE RUNNING
; rung 61
LD H120.02  ; 03ST_STEP 02_WorkPiece Clamp Down Good Condition for other process
OUT 4243.00  ; Workpiece clamp downward signal
; rung 62
LD H120.06  ; 03ST_STEP 06_Measuring Good Condition Signal for other process
OUT 4243.01  ; Measurement strating signal
; rung 63
LD H120.02  ; 03ST_STEP 02_WorkPiece Clamp Down Good Condition for other process
OR H120.03  ; 03ST_STEP 03_Workpiece Clamp Signal Transfer Complet
OR H120.04  ; 03ST_STEP 04_Waiting WorkPiece Clam Down Complete
OR H120.05  ; 03ST_STEP 05_Transfer Carrier Up
OR H120.06  ; 03ST_STEP 06_Measuring Good Condition Signal for other process
OUT 4243.10  ; TRANSFER CARRIER FORWARD
; rung 64
LD H120.09  ; 03ST_STEP 09
OUT 4243.02  ; Transfer-carrier backward signal receipt

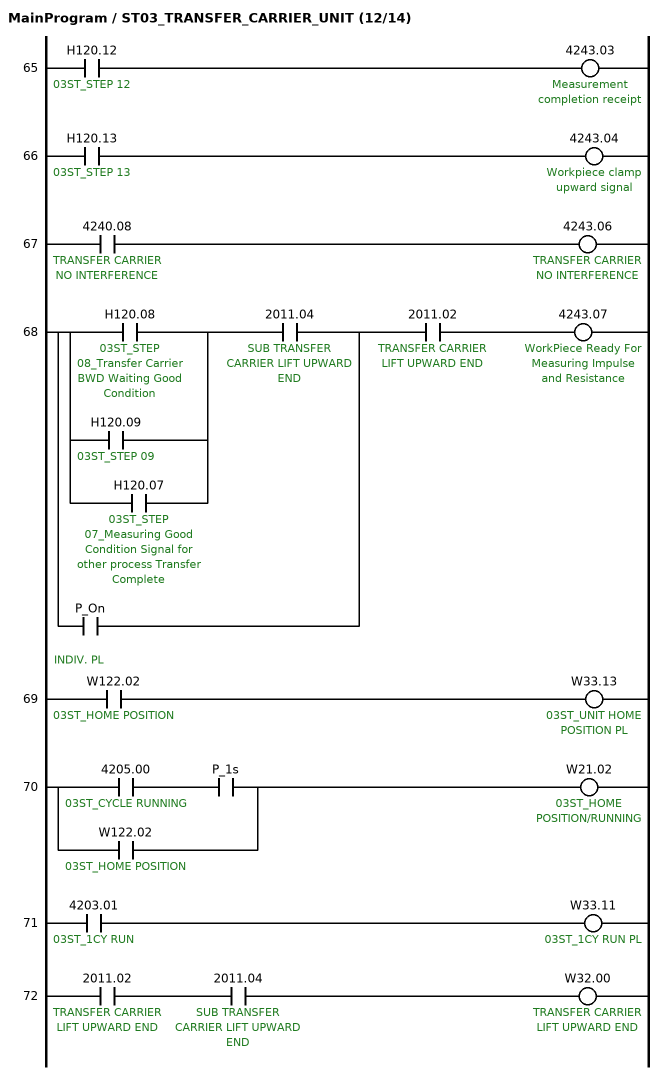
; rung 65
LD H120.12  ; 03ST_STEP 12
OUT 4243.03  ; Measurement completion receipt
; rung 66
LD H120.13  ; 03ST_STEP 13
OUT 4243.04  ; Workpiece clamp upward signal
; rung 67
LD 4240.08  ; TRANSFER CARRIER NO INTERFERENCE
OUT 4243.06  ; TRANSFER CARRIER NO INTERFERENCE
; rung 68
LD H120.08  ; 03ST_STEP 08_Transfer Carrier BWD Waiting Good Condition
OR H120.09  ; 03ST_STEP 09
OR H120.07  ; 03ST_STEP 07_Measuring Good Condition Signal for other process Transfer Complete
AND 2011.04  ; SUB TRANSFER CARRIER LIFT UPWARD END
OR P_On
AND 2011.02  ; TRANSFER CARRIER LIFT UPWARD END
OUT 4243.07  ; WorkPiece Ready For Measuring Impulse and Resistance
; rung 69: INDIV. PL
LD W122.02  ; 03ST_HOME POSITION
OUT W33.13  ; 03ST_UNIT HOME POSITION PL
; rung 70
LD 4205.00  ; 03ST_CYCLE RUNNING
AND P_1s
OR W122.02  ; 03ST_HOME POSITION
OUT W21.02  ; 03ST_HOME POSITION/RUNNING
; rung 71
LD 4203.01  ; 03ST_1CY RUN
OUT W33.11  ; 03ST_1CY RUN PL
; rung 72
LD 2011.02  ; TRANSFER CARRIER LIFT UPWARD END
AND 2011.04  ; SUB TRANSFER CARRIER LIFT UPWARD END
OUT W32.00  ; TRANSFER CARRIER LIFT UPWARD END

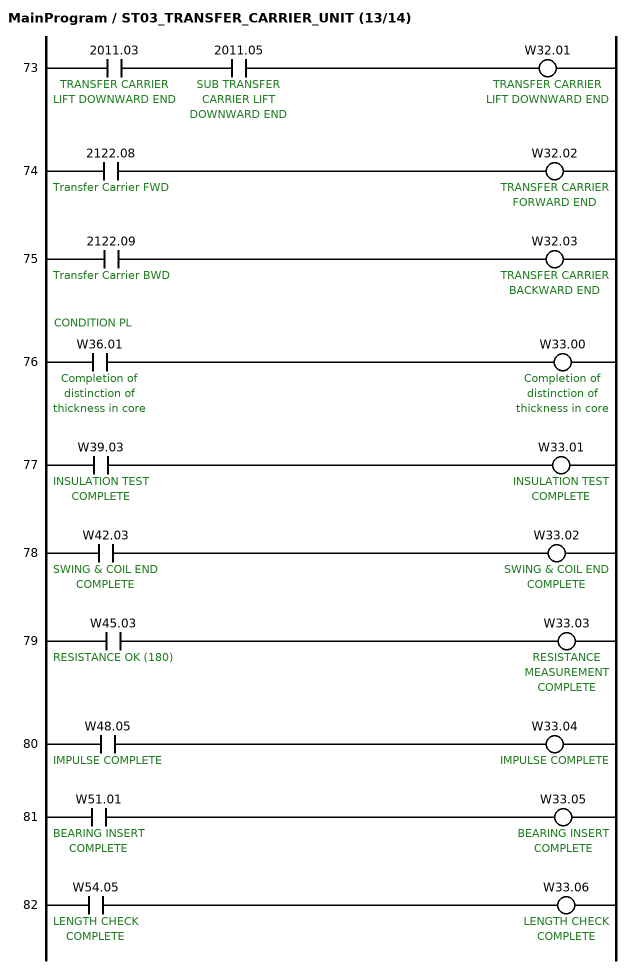
; rung 73
LD 2011.03  ; TRANSFER CARRIER LIFT DOWNWARD END
AND 2011.05  ; SUB TRANSFER CARRIER LIFT DOWNWARD END
OUT W32.01  ; TRANSFER CARRIER LIFT DOWNWARD END
; rung 74
LD 2122.08  ; Transfer Carrier FWD
OUT W32.02  ; TRANSFER CARRIER FORWARD END
; rung 75
LD 2122.09  ; Transfer Carrier BWD
OUT W32.03  ; TRANSFER CARRIER BACKWARD END
; rung 76: CONDITION PL
LD W36.01  ; Completion of distinction of thickness in core
OUT W33.00  ; Completion of distinction of thickness in core
; rung 77
LD W39.03  ; INSULATION TEST COMPLETE
OUT W33.01  ; INSULATION TEST COMPLETE
; rung 78
LD W42.03  ; SWING & COIL END COMPLETE
OUT W33.02  ; SWING & COIL END COMPLETE
; rung 79
LD W45.03  ; RESISTANCE OK (180)
OUT W33.03  ; RESISTANCE MEASUREMENT COMPLETE
; rung 80
LD W48.05  ; IMPULSE COMPLETE
OUT W33.04  ; IMPULSE COMPLETE
; rung 81
LD W51.01  ; BEARING INSERT COMPLETE
OUT W33.05  ; BEARING INSERT COMPLETE
; rung 82
LD W54.05  ; LENGTH CHECK COMPLETE
OUT W33.06  ; LENGTH CHECK COMPLETE

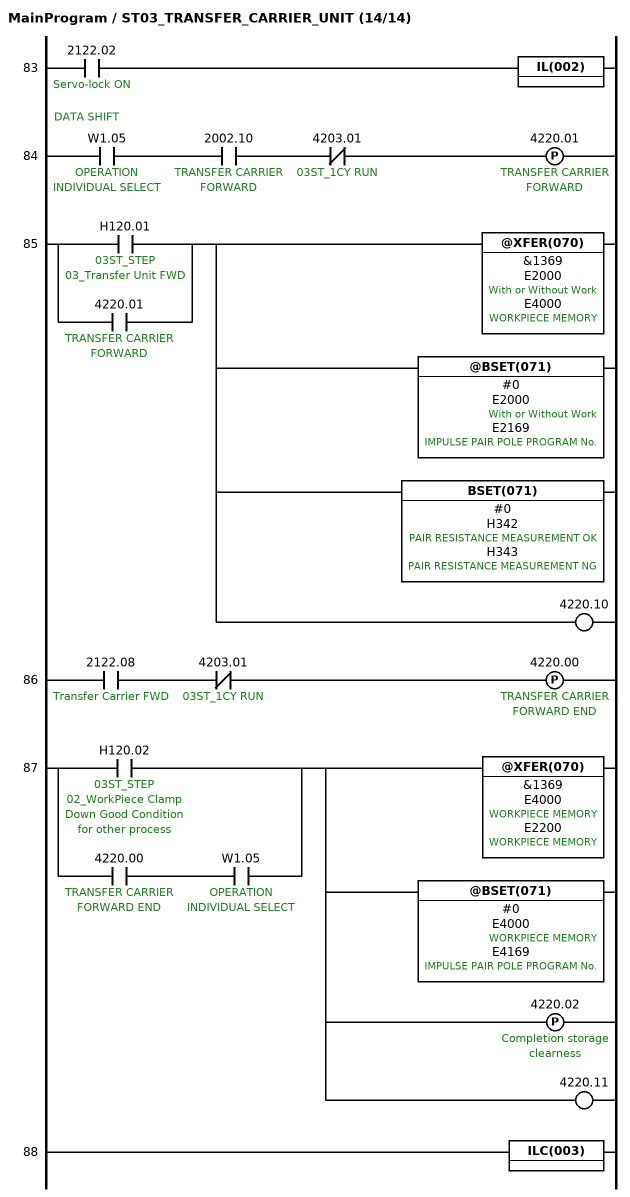
; rung 83
LD 2122.02  ; Servo-lock ON
IL(002)
; rung 84: DATA SHIFT
LD W1.05  ; OPERATION INDIVIDUAL SELECT
AND 2002.10  ; TRANSFER CARRIER FORWARD
ANDNOT 4203.01  ; 03ST_1CY RUN
DIFU(013) 4220.01  ; TRANSFER CARRIER FORWARD
; rung 85
LD H120.01  ; 03ST_STEP 03_Transfer Unit FWD
OR 4220.01  ; TRANSFER CARRIER FORWARD
@XFER(070) &1369 E2000 E4000  ; With or Without Work, WORKPIECE MEMORY
@BSET(071) #0 E2000 E2169  ; With or Without Work, IMPULSE PAIR POLE PROGRAM No.
BSET(071) #0 H342 H343  ; PAIR RESISTANCE MEASUREMENT OK, PAIR RESISTANCE MEASUREMENT NG
OUT 4220.10
; rung 86
LD 2122.08  ; Transfer Carrier FWD
ANDNOT 4203.01  ; 03ST_1CY RUN
DIFU(013) 4220.00  ; TRANSFER CARRIER FORWARD END
; rung 87
LD H120.02  ; 03ST_STEP 02_WorkPiece Clamp Down Good Condition for other process
LD 4220.00  ; TRANSFER CARRIER FORWARD END
AND W1.05  ; OPERATION INDIVIDUAL SELECT
ORLD
@XFER(070) &1369 E4000 E2200  ; WORKPIECE MEMORY
@BSET(071) #0 E4000 E4169  ; WORKPIECE MEMORY, IMPULSE PAIR POLE PROGRAM No.
DIFU(013) 4220.02  ; Completion storage clearness
OUT 4220.11
; rung 88
ILC(003)

### Section ST04_WORKPIECE_PUSHER_UNIT

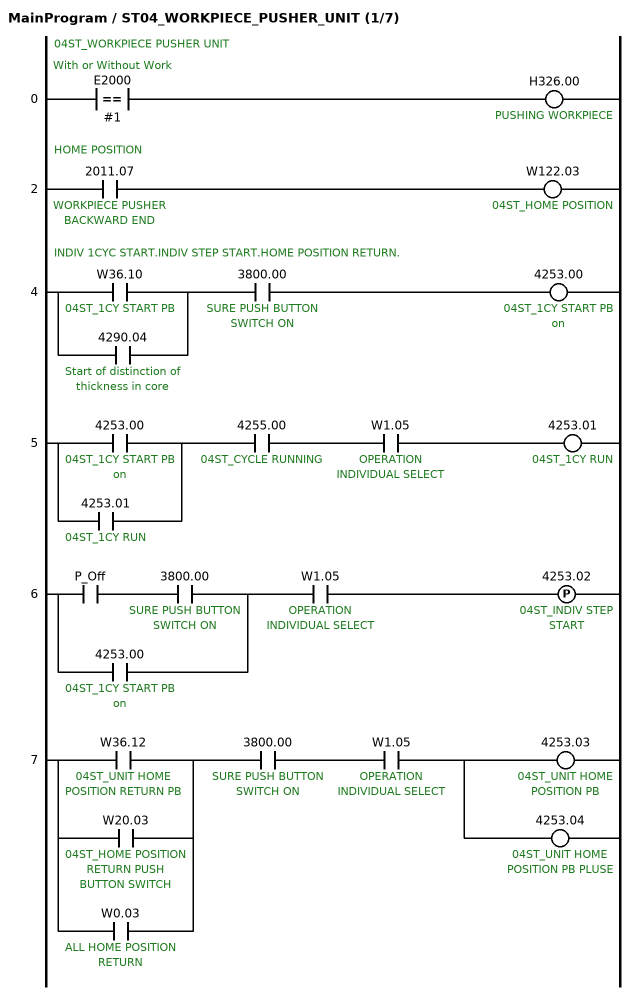
; rung 0: 04ST_WORKPIECE PUSHER UNIT
LD=(300) E2000 #1  ; With or Without Work
OUT H326.00  ; PUSHING WORKPIECE
; rung 1: TIMER
; rung 2: HOME POSITION
LD 2011.07  ; WORKPIECE PUSHER BACKWARD END
OUT W122.03  ; 04ST_HOME POSITION
; rung 3: INTERFERENCE
; rung 4: INDIV 1CYC START.INDIV STEP START.HOME POSITION RETURN.
LD W36.10  ; 04ST_1CY START PB
OR 4290.04  ; Start of distinction of thickness in core
AND 3800.00  ; SURE PUSH BUTTON SWITCH ON
OUT 4253.00  ; 04ST_1CY START PB on
; rung 5
LD 4253.00  ; 04ST_1CY START PB on
OR 4253.01  ; 04ST_1CY RUN
AND 4255.00  ; 04ST_CYCLE RUNNING
AND W1.05  ; OPERATION INDIVIDUAL SELECT
OUT 4253.01  ; 04ST_1CY RUN
; rung 6
LD P_Off
AND 3800.00  ; SURE PUSH BUTTON SWITCH ON
OR 4253.00  ; 04ST_1CY START PB on
AND W1.05  ; OPERATION INDIVIDUAL SELECT
DIFU(013) 4253.02  ; 04ST_INDIV STEP START
; rung 7
LD W36.12  ; 04ST_UNIT HOME POSITION RETURN PB
OR W20.03  ; 04ST_HOME POSITION RETURN PUSH BUTTON SWITCH
OR W0.03  ; ALL HOME POSITION RETURN
AND 3800.00  ; SURE PUSH BUTTON SWITCH ON
AND W1.05  ; OPERATION INDIVIDUAL SELECT
OUT 4253.03  ; 04ST_UNIT HOME POSITION PB
OUT 4253.04  ; 04ST_UNIT HOME POSITION PB PLUSE

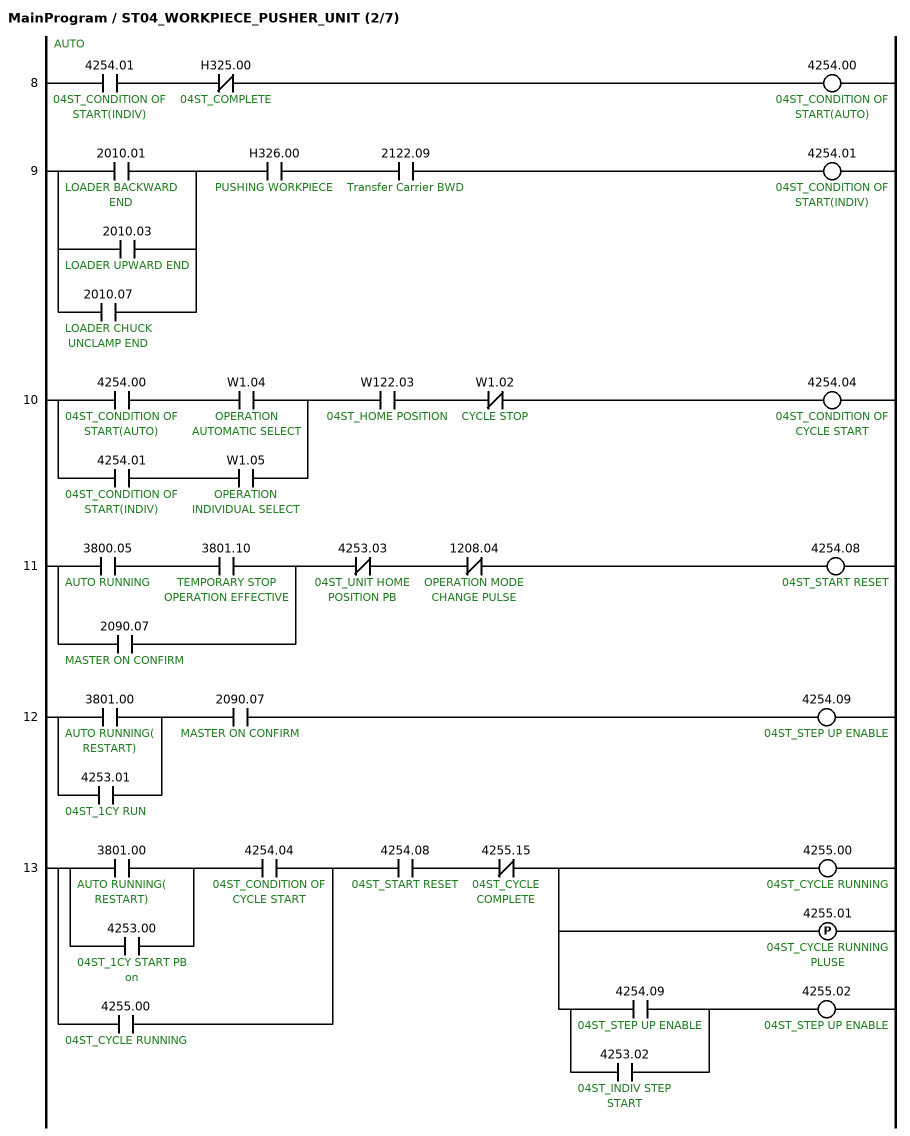
; rung 8: AUTO
LD 4254.01  ; 04ST_CONDITION OF START(INDIV)
ANDNOT H325.00  ; 04ST_COMPLETE
OUT 4254.00  ; 04ST_CONDITION OF START(AUTO)
; rung 9
LD 2010.01  ; LOADER BACKWARD END
OR 2010.03  ; LOADER UPWARD END
OR 2010.07  ; LOADER CHUCK UNCLAMP END
AND H326.00  ; PUSHING WORKPIECE
AND 2122.09  ; Transfer Carrier BWD
OUT 4254.01  ; 04ST_CONDITION OF START(INDIV)
; rung 10
LD 4254.00  ; 04ST_CONDITION OF START(AUTO)
AND W1.04  ; OPERATION AUTOMATIC SELECT
LD 4254.01  ; 04ST_CONDITION OF START(INDIV)
AND W1.05  ; OPERATION INDIVIDUAL SELECT
ORLD
AND W122.03  ; 04ST_HOME POSITION
ANDNOT W1.02  ; CYCLE STOP
OUT 4254.04  ; 04ST_CONDITION OF CYCLE START
; rung 11
LD 3800.05  ; AUTO RUNNING
AND 3801.10  ; TEMPORARY STOP OPERATION EFFECTIVE
OR 2090.07  ; MASTER ON CONFIRM
ANDNOT 4253.03  ; 04ST_UNIT HOME POSITION PB
ANDNOT 1208.04  ; OPERATION MODE CHANGE PULSE
OUT 4254.08  ; 04ST_START RESET
; rung 12
LD 3801.00  ; AUTO RUNNING(RESTART)
OR 4253.01  ; 04ST_1CY RUN
AND 2090.07  ; MASTER ON CONFIRM
OUT 4254.09  ; 04ST_STEP UP ENABLE
; rung 13
LD 3801.00  ; AUTO RUNNING(RESTART)
OR 4253.00  ; 04ST_1CY START PB on
AND 4254.04  ; 04ST_CONDITION OF CYCLE START
OR 4255.00  ; 04ST_CYCLE RUNNING
AND 4254.08  ; 04ST_START RESET
ANDNOT 4255.15  ; 04ST_CYCLE COMPLETE
OUT 4255.00  ; 04ST_CYCLE RUNNING
DIFU(013) 4255.01  ; 04ST_CYCLE RUNNING PLUSE
LD 4254.09  ; 04ST_STEP UP ENABLE
OR 4253.02  ; 04ST_INDIV STEP START
ANDLD
OUT 4255.02  ; 04ST_STEP UP ENABLE

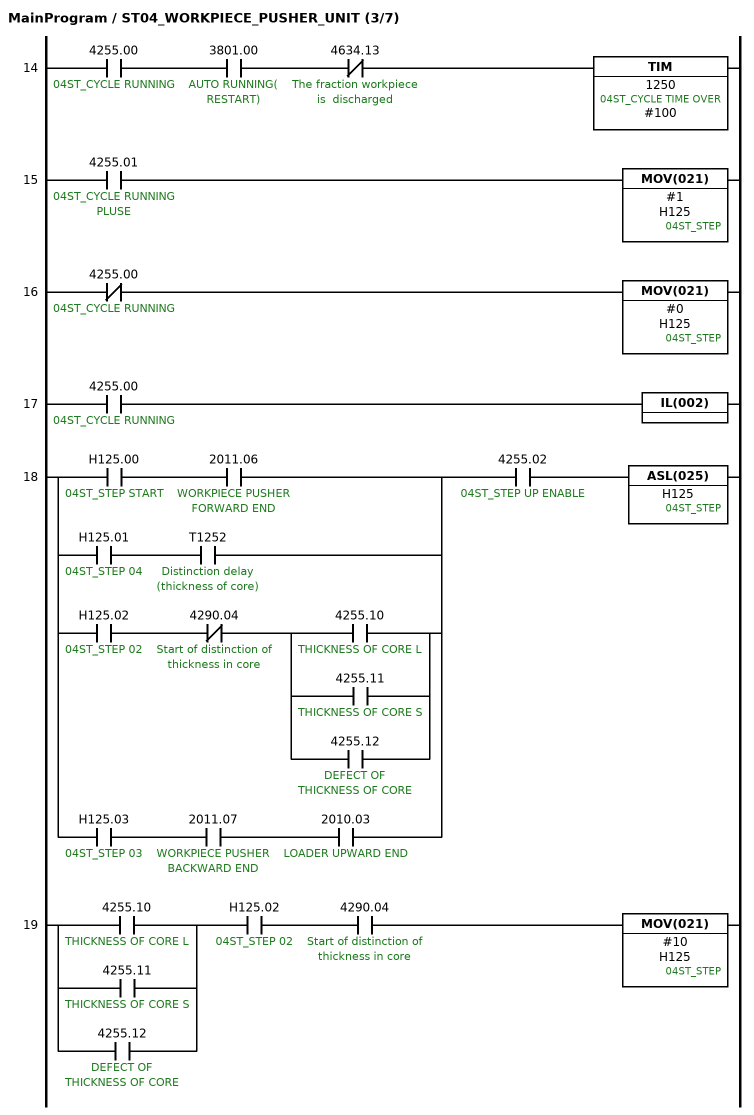
; rung 14
LD 4255.00  ; 04ST_CYCLE RUNNING
AND 3801.00  ; AUTO RUNNING(RESTART)
ANDNOT 4634.13  ; The fraction workpiece is  discharged
TIM 1250 #100  ; 04ST_CYCLE TIME OVER
; rung 15
LD 4255.01  ; 04ST_CYCLE RUNNING PLUSE
MOV(021) #1 H125  ; 04ST_STEP
; rung 16
LDNOT 4255.00  ; 04ST_CYCLE RUNNING
MOV(021) #0 H125  ; 04ST_STEP
; rung 17
LD 4255.00  ; 04ST_CYCLE RUNNING
IL(002)
; rung 18
LD H125.00  ; 04ST_STEP START
AND 2011.06  ; WORKPIECE PUSHER FORWARD END
LD H125.01  ; 04ST_STEP 04
AND T1252  ; Distinction delay (thickness of core)
ORLD
LD H125.02  ; 04ST_STEP 02
ANDNOT 4290.04  ; Start of distinction of thickness in core
LD 4255.10  ; THICKNESS OF CORE L
OR 4255.11  ; THICKNESS OF CORE S
OR 4255.12  ; DEFECT OF THICKNESS OF CORE
ANDLD
ORLD
LD H125.03  ; 04ST_STEP 03
AND 2011.07  ; WORKPIECE PUSHER BACKWARD END
AND 2010.03  ; LOADER UPWARD END
ORLD
AND 4255.02  ; 04ST_STEP UP ENABLE
ASL(025) H125  ; 04ST_STEP
; rung 19
LD 4255.10  ; THICKNESS OF CORE L
OR 4255.11  ; THICKNESS OF CORE S
OR 4255.12  ; DEFECT OF THICKNESS OF CORE
AND H125.02  ; 04ST_STEP 02
AND 4290.04  ; Start of distinction of thickness in core
MOV(021) #10 H125  ; 04ST_STEP

